(* Logix 5000 project; controller VET 1756-L62 rev 19.52; software revision 19.01 *)

TASK DB (periodic, rate 500 ms, priority 10, watchdog 500 ms) : Main
TASK Dosificador (periodic, rate 40 ms, priority 10, watchdog 250 ms) : Dosificar_MAC_01, Dosificar_MID_01, Dosificar_MIC_01
TASK DRT (periodic, rate 50 ms, priority 1, watchdog 500 ms) : _Ctrl_drt
TASK MainTask (periodic, rate 50 ms, priority 5, watchdog 500 ms) : Main1, Gestion_Dosificacion
TASK Typlgie (periodic, rate 400 ms, priority 10, watchdog 900 ms) : Typlgie

MODULES
   Local : 1756-L62 (ICP 12, rev 19.52)
END_MODULES

TYPE batch :
STRUCT
   Head : batch_cabecera;
   Data : batch_detalle;
END_STRUCT
END_TYPE

TYPE batch_cabecera :
STRUCT
   folio : DINT;
   orden : DINT;
   formula : SHORTSTRING;
   estado : SINT;
   correlativo : SINT;
   total_batch : SINT;
   peso_teorico : REAL;
   flags : SINT;
END_STRUCT
END_TYPE

TYPE batch_detalle :
STRUCT
   codigo : INT[40];   // Código Ingrediente
   peso_f : REAL[40];   // Peso Formula
   peso_r : REAL[40];   // Peso Real
   tolva : SINT[40];   // Tolva Utilizada
   lugar : SINT[40];   // Lugar donde Dosificar
   flags : SINT[40];   // Flags
   fecha_i : DINT[40];
   fecha_f : DINT[40];
   hora_i : DINT[40];
   hora_f : DINT[40];
END_STRUCT
END_TYPE

TYPE Bins_Setup :
STRUCT
   c : tabbin_head;
   d : tabbin_data[2];
END_STRUCT
END_TYPE

TYPE cola_almacenes :
STRUCT
   origen : DINT;
   destino : DINT;
   cantidad : REAL;
   folio_op : DINT;
   fecha : DINT;
   hora : DINT;
END_STRUCT
END_TYPE

TYPE comandos_eph :
STRUCT
   start : BOOL;
   hold : BOOL;
   restart : BOOL;
   stop : BOOL;
   abort : BOOL;
   reset : BOOL;
   reset_especial : BOOL;
END_STRUCT
END_TYPE

TYPE dosif_struct :
STRUCT
   peso_terreno : REAL;
   frq_terreno : REAL;
   idx_ing : INT;
   idx_batch : INT;
   msg : DINT;
   ans : DINT;
   resultado : INT;
   estado_phases : estado_eph;
   comandos_phases : comandos_eph;
END_STRUCT
END_TYPE

TYPE DRTs :   // Estructura para DRT
STRUCT
   InputPos : DINT;   // Posicion Leida (Bits)
   CmdPos : DINT;   // Posicion Comanda
   ConfPos : DINT;   // Posicion Confirmada
   RealPos : DINT;   // Posicion Leida (Num)
   TotalPos : DINT;   // Total Posiciones
END_STRUCT
END_TYPE

TYPE Eqp_Bits :
STRUCT
   Bits1 : DINT;
   Bits2 : DINT;
   Bits3 : DINT;
   Bits4 : DINT;
END_STRUCT
END_TYPE

TYPE Eqp_Cfg :
STRUCT
   Type : DINT;   // Eqp Type
   Setup : DINT;   // Config
   Syst : DINT;   // System Group
   Plant : DINT;   // Plant
   Prst1 : DINT;   // Preset Timer1
   Prst2 : DINT;   // Preset Timer2
   Prst3 : DINT;   // Preset Timer3
   Prst4 : DINT;   // Preset Timer4
   Prst5 : DINT;   // Preset Timer5
   Prst6 : DINT;   // Preset Timer6
END_STRUCT
END_TYPE

TYPE Eqp_Timers :
STRUCT
   Tpo1 : TIMER;
   Tpo2 : TIMER;
   Tpo3 : TIMER;
   Tpo4 : TIMER;
   Tpo5 : TIMER;
   Tpo6 : TIMER;
END_STRUCT
END_TYPE

TYPE Eqp_Typologie :
STRUCT
   Next : DINT;
   Type : DINT;
   Setup : DINT;
   Syst : DINT;
   Area : DINT;
   Indx : DINT[16];
END_STRUCT
END_TYPE

TYPE Equipo :
STRUCT
   Timer : Eqp_Timers;   // Equipment Timers
   S : Eqp_Bits;
   Next : DINT;
   Color : DINT;
END_STRUCT
END_TYPE

TYPE estado_eph :
STRUCT
   _aborted : BOOL;   // Estado Aborted
   _held : BOOL;   // Estado Held
   _idle : BOOL;   // Estado Idle
   _running : BOOL;   // Estado Running
   _complete : BOOL;   // Estado Complete
   _stopped : BOOL;   // Estado Stopped
END_STRUCT
END_TYPE

TYPE falla_aux :
STRUCT
   Time_Low : DINT;
   Time_High : DINT;
   Type : INT;
   Code : INT;
   Info : DINT[8];
   Falla : BOOL;
END_STRUCT
END_TYPE

TYPE Fault_Register :   // Almacena el valor de MAJORFAULTRECORD
STRUCT
   Time_Low : DINT;
   Time_High : DINT;
   Type : INT;
   Code : INT;
   Info : DINT[8];
END_STRUCT
END_TYPE

TYPE flujometro :   // Manejo de Flujometros
STRUCT
   scale_flujo : ScaleAIO;
   scale_total : ScaleAIO;
   flujo : REAL;   // Flujo
   total : REAL;   // Total sin Escalamiento
   total_batch : REAL;   // Peso sin Escalamiento x Batch
   total_scaled : REAL;   // Peso Escalado
   total_scaled_batch : REAL;   // Peso Escalado x Batch
   T : TIMER;
   set_in : REAL;   // Escalamiento Peso Entrada
   set_out : REAL;   // Escalamiento Peso Salida
   aux : DINT;   // Usos Varios
   input : DINT;   // Entrada desde flujómetro
   delta_t : DINT;   // Variación de tiempo en mseg desde la medición anterior
END_STRUCT
END_TYPE

TYPE Index :
STRUCT
   a : DINT;
   b : DINT;
   c : DINT;
   d : DINT;
   e : DINT;
   f : DINT;
   g : DINT;
   h : DINT;
   i : DINT;
   j : DINT;
   k : DINT;
   l : DINT;
   m : DINT;
   n : DINT;
   o : DINT;
   p : DINT;
   q : DINT;
   r : DINT;
   s : DINT;
   t : DINT;
   u : DINT;
   v : DINT;
   w : DINT;
   x : DINT;
   y : DINT;
   z : DINT;
   a1 : DINT;
   b1 : DINT;
   c1 : DINT;
   d1 : DINT;
   e1 : DINT;
   f1 : DINT;
   g1 : DINT;
   h1 : DINT;
   i1 : DINT;
   j1 : DINT;
   k1 : DINT;
   l1 : DINT;
   m1 : DINT;
   n1 : DINT;
   o1 : DINT;
   p1 : DINT;
   q1 : DINT;
   r1 : DINT;
   s1 : DINT;
   t1 : DINT;
   u1 : DINT;
   v1 : DINT;
   w1 : DINT;
   x1 : DINT;
   y1 : DINT;
   z1 : DINT;
   a2 : DINT;
   b2 : DINT;
   c2 : DINT;
   d2 : DINT;
   e2 : DINT;
   f2 : DINT;
   g2 : DINT;
   h2 : DINT;
   i2 : DINT;
   j2 : DINT;
   k2 : DINT;
   l2 : DINT;
   m2 : DINT;
   n2 : DINT;
   o2 : DINT;
   p2 : DINT;
   q2 : DINT;
   r2 : DINT;
   s2 : DINT;
   t2 : DINT;
   u2 : DINT;
   v2 : DINT;
   w2 : DINT;
   x2 : DINT;
   y2 : DINT;
   z2 : DINT;
   a3 : DINT;
   b3 : DINT;
   c3 : DINT;
   d3 : DINT;
   e3 : DINT;
   f3 : DINT;
   g3 : DINT;
   h3 : DINT;
   i3 : DINT;
   j3 : DINT;
   k3 : DINT;
   l3 : DINT;
   m3 : DINT;
   n3 : DINT;
   o3 : DINT;
   p3 : DINT;
   q3 : DINT;
   r3 : DINT;
   s3 : DINT;
   t3 : DINT;
   u3 : DINT;
   v3 : DINT;
   w3 : DINT;
   x3 : DINT;
   y3 : DINT;
   z3 : DINT;
END_STRUCT
END_TYPE

TYPE Origen :
STRUCT
   Index : DINT;   // Index
   _1eqp : DINT;   // Indice Primer Equipo
   Bits : DINT;
   Color : INT;   // Color Linea
   DestReal : DINT;   // Indice Equipo Destino Final Real
   DestOld : DINT;   // Indice Equipo Destino Final Real Old
   DestNew : INT;   // Sub Indice Destino Final
   Prod1eqpInd : DINT;   // Indice Producto Primer Equipo
   ProdFinInd : DINT;   // Indice Producto Bin Final
   Prod1eqp : DINT;   // Codigo Producto Primer Equipo
   ProdFin : DINT;   // Codigo Producto Bin Final
   State : DINT;   // Estado
   Tespera : TIMER;   // Si se cumple este tiempo y no ha partido la ruta se quita la OMR
END_STRUCT
END_TYPE

TYPE PID_Info :
STRUCT
   PV : DINT;   // Process Variable (0-100%)
   SP : DINT;   // Setpoint (0-100%)
   CV : DINT;   // Control Variable (0-100%)
END_STRUCT
END_TYPE

TYPE PID_Struct :
STRUCT
   Core : PID;   // PID Core Instruction
   Status : DINT;   // Status Bits
   Info : PID_Info;   // Extra Information
   PV : REAL;   // Process Variable (ENU)
   SP : REAL;   // Setpoint (ENU)
   CV : REAL;   // Control Variable (0-100%)
   DB : REAL;   // Deadband (ENU)
   Upd : REAL;   // Loop Update Time (sec)
   Kp : REAL;   // Proportional Gain
   Ki : REAL;   // Integral Gain (1/sec)
   Kd : REAL;   // Derivative Time (sec)
   ENU_LL : REAL;   // ENU Low Limit
   ENU_LH : REAL;   // ENU High Limit
   AI : DINT;   // PV - Analog Input (0-4095)
   AO : DINT;   // CV - Analog Output (0-4095)
END_STRUCT
END_TYPE

TYPE Sel_eqp :   // Equipos pertenecientes a selectores
STRUCT
   IDX_SEL : INT;   // Indice Selector al que pertenece
   IDX_EQP : INT;   // Indice Equipo en Tabla Equipos
   POS_CMD : SINT[32];   // Comandos segun posicion
END_STRUCT
END_TYPE

TYPE Selector :
STRUCT
   Idx_eqp : INT;   // Indice en Tabla Equipo
   Next : INT[32];   // Siguiente segun posicion
   Pos_Conf : SINT;   // Posicion Confirmada
   Pos_Cmd : SINT;   // Posicion Comandada
   Pos_Real : SINT;   // Posicion Leida equipos
   Pos_Old : SINT;   // Posicion Anterior RSV
   Pos_New : SINT;   // Posicion Nueva RSV
   Pos_Fut : SINT;   // Posicion Futura RSV
   Pos_Cant : SINT;   // Cantidad de Posiciones
   Pos_CM : SINT;   // Posicion con conf. de marcha
   Idx_1Tabeqp : INT;   // Idx 1er eqp en Tabeqp
   Timer1 : TIMER;
   Timer2 : TIMER;
END_STRUCT
END_TYPE

TYPE set_variables :
STRUCT
   D : DINT[50];
   F : REAL[40];
   T : TIMER[10];
   setD : DINT[10];
   SetF : REAL[10];
   i0 : DINT;
   i1 : DINT;
   i2 : DINT;
   i3 : DINT;
   i4 : DINT;
   i5 : DINT;
   i6 : DINT;
   i7 : DINT;
   i8 : DINT;
   i9 : DINT;
   i10 : DINT;
   i11 : DINT;
   i12 : DINT;
   i13 : DINT;
   i14 : DINT;
   i15 : DINT;
   i16 : DINT;
   i17 : DINT;
   i18 : DINT;
   i19 : DINT;
END_STRUCT
END_TYPE

TYPE SHORTSTRING :
STRUCT
   LEN : DINT;
   DATA : SINT[10];
END_STRUCT
END_TYPE

TYPE Soft_Starter :
STRUCT
   Idx_Equipo : DINT[10];
   Eqp_Actual : DINT;
   Partiendo : BOOL;
   Esperando : BOOL;
   Disponible : BOOL;
   Flags : DINT;
   Procesando : BOOL;
   Tpo_Espera : TIMER;
   Tpos_Grl : TIMER[2];
END_STRUCT
END_TYPE

TYPE STRING12 :
STRUCT
   LEN : DINT;
   DATA : SINT[12];
END_STRUCT
END_TYPE

TYPE STRING14 :
STRUCT
   LEN : DINT;
   DATA : SINT[14];
END_STRUCT
END_TYPE

TYPE Tab_O_D_Dest :
STRUCT
   D : Tab_O_D_Sel[30];   // Destinos Posibles
   Eqp : INT[30];
END_STRUCT
END_TYPE

TYPE Tab_O_D_Orig :
STRUCT
   O : Tab_O_D_Dest[13];   // Numero de Orígnes
END_STRUCT
END_TYPE

TYPE Tab_O_D_Sel :
STRUCT
   S : INT[10];   // NUmero de Selectores
END_STRUCT
END_TYPE

TYPE tabbin_data :
STRUCT
   t_espera : INT[80];   // Tiempo Espera (mSeg)
   t_pulso : INT[80];   // Tiempo Ajuste (mSeg)
   precorte : REAL[80];   // Precorte
   error_per : REAL[80];   // Error Permitido (%)
   error_kg : REAL[80];   // Error Permitido (Kg)
   frec_inicial : REAL[80];   // Frecuencia A (Hz)
   frec_final : REAL[80];   // Frecuencia B (Hz)
   curvatura : REAL[80];   // Curvatura exponencial
   porcentaje_frec_max : REAL[80];   // Porcentaje del peso de detención con dosificación a frecuencia máxima
   low_limit : REAL[80];   // Límite Inferior
   high_limit : REAL[80];   // Límite Superior
   flags : DINT[80];   // Flags Varios
END_STRUCT
END_TYPE

TYPE tabbin_head :
STRUCT
   id : SINT[80];   // Identificador Único de tolva (Correlativo)
   tolva : INT[80];   // Número de Tolva
   n_tolva : DINT[80];   // Número de equipo de la tolva
   equipo1 : INT[80];   // Equipo dosificador
   equipo2 : INT[80];   // Equipo dosificador
   equipo3 : INT[80];   // Equipo dosificador
   equipo4 : INT[80];   // Equipo dosificador
   equipo5 : INT[80];   // Equipo dosificador
   dosificador : INT[80];
   codigo : DINT[80];   // Codigo Ingrediente
   sql_codigo : DINT[80];   // Codigo desde Oracle
   prioridad : INT[80];   // Prioridad
   nivel_bajo : DINT[80];
   nivel_alto : DINT[80];
   tipo : INT[80];
   ind_peso : INT[80];
END_STRUCT
END_TYPE

TYPE tabDosif :   // Tabla de Dosificadores
STRUCT
   idx_tolva : DINT[20];
   idx_vdf : DINT[20];
   idx_flujometro : DINT[20];
   tipo : DINT[20];
END_STRUCT
END_TYPE

TYPE variables_procedimientos :
STRUCT
   step_idx : INT;
   trigger : SINT[5];
   handshake : SINT[5];
   in_tstamp : DINT[5];
   out_tstamp : DINT[5];
   out_res : SINT[5];
   D : DINT[10];
   F : REAL[5];
   i0 : INT;
   i1 : INT;
   i2 : INT;
   i3 : INT;
   i4 : INT;
   SetD : DINT[3];
   SetF : DINT[3];
   T : TIMER[10];
END_STRUCT
END_TYPE

TYPE variables_sproc :
STRUCT
   step_idx : DINT;
   trigger : DINT[3];
   handshake : DINT[3];
   in_tstamp : DINT[3];
   out_tstamp : DINT[3];
   out_res : DINT[3];
   D : DINT[10];
   F : REAL[5];
   i0 : DINT;
   i1 : DINT;
   i2 : DINT;
   i3 : DINT;
   i4 : DINT;
   SetD : DINT[3];
   SetF : DINT[3];
   T : TIMER[5];
END_STRUCT
END_TYPE

TYPE VDFS :
STRUCT
   ST : DINT;
   CMD : DINT;
   FRQ_IN : REAL;
   FRQ_OUT : REAL;
   I : REAL;
   P : REAL;
   V : REAL;
   AUX : DINT[5];
   SCALE : ScaleAIO[2];
   Sincro_MSG : SINT;
END_STRUCT
END_TYPE

ADD_ON_INSTRUCTION ScaleAIO   (* revision 1.0, vendor Ole Bank *)
VAR_INPUT
   Input : REAL; {required}
   InLow : REAL; {required}
   InHigh : REAL; {required}
   OutLow : REAL; {required}
   OutHigh : REAL; {required}
END_VAR
VAR_OUTPUT
   Output : REAL; {access Read Only, required}
END_VAR

ROUTINE Logic   (* ladder *)
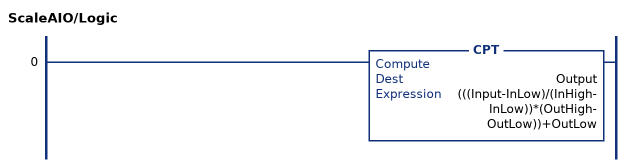
   0: CPT(Output,(((Input-InLow)/(InHigh-InLow))*(OutHigh-OutLow))+OutLow);
END_ROUTINE
END_ADD_ON_INSTRUCTION

ADD_ON_INSTRUCTION velocidad_exp   (* revision 1.0 *)
VAR_INPUT
   x : REAL; {required}
   curvatura : REAL; {required}
   V_inicial : REAL; {required}
   V_final : REAL; {required}
END_VAR
VAR_OUTPUT
   V_salida : REAL; {access Read Only, required}
END_VAR

ROUTINE Logic   (* ladder *)
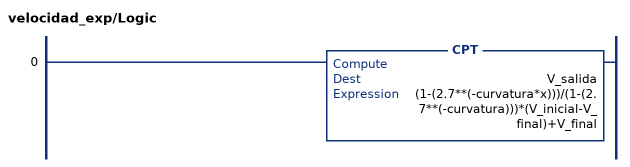
   0: CPT(V_salida,(1-(2.7**(-curvatura*x)))/(1-(2.7**(-curvatura)))*(V_inicial-V_final)+V_final);
END_ROUTINE
END_ADD_ON_INSTRUCTION

VAR_GLOBAL   (* controller tags *)
   _BatCode : DINT[100] := ([0] := 22, [1] := 27, [6] := 17, [28] := 171903600, [29] := 171903600, [30] := 96, [31] := 190628600, [32] := 171680000, [33] := 171903600, [34] := 190628600, [35] := 822086000, [36] := 369524000, [40] := 375774000, [41] := 375774000, [42] := 781952000, [70] := 96);
        [20]   // Codigo DOsificación Macros
        [21]   // Cod. Tolva bajo tolvas pesaje macros
        [31]   // TOL-102-00 Batch
        [32]   // TOL-103-00 Batch
        [33]   // TOL-109-00 Batch
        [34]   // TOL-113-00 Batch
        [36]   // TOL-115-00 Batch
   _Codes : DINT[500] := ([1] := 51, [2] := 51, [3] := 51, [4] := 51, [5] := 51, [6] := 51, [7] := 51, [8] := 51, [9] := 51, [10] := 51, [11] := 51, [12] := 51, [13] := 51, [14] := 51, [15] := 51, [16] := 51, [17] := 51, [18] := 51, [19] := 51, [20] := 51, [21] := 70, [22] := 71, [23] := 72, [24] := 73, [26] := 74, [27] := 75, [28] := 76, [29] := 77, [30] := 78, [31] := 79, [32] := 80, [38] := 81, [101] := 1, [102] := 2, [103] := 3, [104] := 4, [111] := 2, [113] := 2, [200] := 7, [201] := 2238, [202] := 7, [203] := 2081, [204] := 2081, [205] := 2081, [206] := 23, [207] := 23, [209] := 23, [210] := 21, [212] := 23, [214] := 7, [301] := 6706, [302] := 6699, [303] := 6706, [304] := 6707, [305] := 6704, [306] := 6706, [307] := 6703, [309] := 6521, [312] := 6670, [315] := 6675,
        [316] := 6707);
   _Eqp : Equipo[800] := ([1].Timer.Tpo1.PRE := 5000, [1].Timer.Tpo2.PRE := 5000, [1].Timer.Tpo3.PRE := 3000, [1].Timer.Tpo4.PRE := 10000, [1].Timer.Tpo5.PRE := 3000, [1].Timer.Tpo6.PRE := 3000, [1].S.Bits1 := 1, [1].S.Bits2 := 495616, [2].Timer.Tpo1.PRE := 5000, [2].Timer.Tpo2.PRE := 5000, [2].Timer.Tpo3.PRE := 3000, [2].Timer.Tpo4.PRE := 10000, [2].Timer.Tpo5.PRE := 3000, [2].Timer.Tpo6.PRE := 3000, [2].S.Bits1 := 4, [2].S.Bits2 := 1409024, [2].S.Bits3 := 16, [3].Timer.Tpo1.PRE := 5000, [3].Timer.Tpo2.PRE := 5000, [3].Timer.Tpo3.PRE := 3000, [3].Timer.Tpo4.PRE := 10000, [3].Timer.Tpo4.ACC := 10027, [3].Timer.Tpo5.PRE := 3000, [3].Timer.Tpo6.PRE := 3000, [3].S.Bits1 := 65, [3].S.Bits2 := 495616, [3].S.Bits3 := 1073807360, [3].Next := 4, [3].Color := 2, [4].Timer.Tpo1.PRE := 5000, [4].Timer.Tpo2.PRE := 5000, [4].Timer.Tpo3.PRE := 3000, [4].Timer.Tpo4.PRE := 10000, [4].Timer.Tpo4.ACC := 10011, [4].Timer.Tpo5.PRE := 3000, [4].Timer.Tpo6.PRE := 3000, [4].S.Bits1 := 81, [4].S.Bits2 := 2600960, [4].S.Bits3 := 1073807361, [4].Next := 170, [4].Color := 2, [5].Timer.Tpo1.PRE := 5000, [5].Timer.Tpo2.PRE := 5000, [5].Timer.Tpo3.PRE := 3000, [5].Timer.Tpo4.PRE := 10000, [5].Timer.Tpo5.PRE := 3000, [5].Timer.Tpo6.PRE := 3000, [5].S.Bits1 := 1, [5].S.Bits2 := 495616, [6].Timer.Tpo1.PRE := 5000, [6].Timer.Tpo2.PRE := 5000, [6].Timer.Tpo3.PRE := 3000, [6].Timer.Tpo4.PRE := 10000, [6].Timer.Tpo5.PRE := 3000, [6].Timer.Tpo6.PRE := 3000, [6].S.Bits1 := 517, [6].S.Bits2 := 69701635, [7].Timer.Tpo1.PRE := 15000, [7].Timer.Tpo2.PRE := 15000, [7].Timer.Tpo3.PRE := 15000,
        [7].Timer.Tpo4.PRE := 20000, [7].Timer.Tpo5.PRE := 1000, [7].Timer.Tpo6.PRE := 1000, [7].S.Bits1 := 19505, [7].S.Bits2 := 2592768, [8].Timer.Tpo1.PRE := 15000, [8].Timer.Tpo2.PRE := 15000, [8].Timer.Tpo3.PRE := 15000, [8].Timer.Tpo4.PRE := 20000, [8].Timer.Tpo5.PRE := 1000, [8].Timer.Tpo6.PRE := 1000, [8].S.Bits1 := 19505, [8].S.Bits2 := 2592768, [9].Timer.Tpo1.PRE := 5000, [9].Timer.Tpo2.PRE := 5000, [9].Timer.Tpo3.PRE := 3000, [9].Timer.Tpo4.PRE := 10000, [9].Timer.Tpo5.PRE := 3000, [9].Timer.Tpo6.PRE := 3000, [10].Timer.Tpo1.PRE := 10000, [10].Timer.Tpo2.PRE := 10000, [10].Timer.Tpo3.PRE := 10000, [10].Timer.Tpo4.PRE := 10000, [10].Timer.Tpo5.PRE := 3000, [10].Timer.Tpo6.PRE := 3000, [10].S.Bits1 := 593, [10].S.Bits2 := 2600960, [10].S.Bits3 := 1073807361, [10].Next := 110, [10].Color := 2, [11].Timer.Tpo1.PRE := 5000, [11].Timer.Tpo2.PRE := 5000, [11].Timer.Tpo3.PRE := 3000, [11].Timer.Tpo4.PRE := 10000, [11].Timer.Tpo5.PRE := 3000, [11].Timer.Tpo6.PRE := 3000, [11].S.Bits1 := 593, [11].S.Bits2 := 2600960, [11].S.Bits3 := 1073807361, [11].Next := 112, [11].Color := 2, [12].Timer.Tpo1.PRE := 5000, [12].Timer.Tpo2.PRE := 5000, [12].Timer.Tpo3.PRE := 3000, [12].Timer.Tpo4.PRE := 45000, [12].Timer.Tpo5.PRE := 15000, [12].Timer.Tpo6.PRE := 3000, [12].S.Bits1 := 593, [12].S.Bits2 := 2600960, [12].S.Bits3 := 1073807361, [12].Next := 112, [12].Color := 2, [13].Timer.Tpo1.PRE := 5000, [13].Timer.Tpo2.PRE := 5000, [13].Timer.Tpo3.PRE := 3000, [13].Timer.Tpo4.PRE := 10000, [13].Timer.Tpo5.PRE := 3000, [13].Timer.Tpo6.PRE := 3000, [13].S.Bits1 := 593, [13].S.Bits2 := 2600960,
        [13].S.Bits3 := 1073807361, [13].Next := 110, [13].Color := 2, [14].Timer.Tpo1.PRE := 5000, [14].Timer.Tpo2.PRE := 5000, [14].Timer.Tpo3.PRE := 3000, [14].Timer.Tpo4.PRE := 10000, [14].Timer.Tpo5.PRE := 3000, [14].Timer.Tpo6.PRE := 3000, [14].S.Bits1 := 593, [14].S.Bits2 := 2600960, [14].S.Bits3 := 1073807361, [14].Next := 110, [14].Color := 2, [15].Timer.Tpo1.PRE := 5000, [15].Timer.Tpo2.PRE := 5000, [15].Timer.Tpo3.PRE := 3000, [15].Timer.Tpo4.PRE := 10000, [15].Timer.Tpo5.PRE := 3000, [15].Timer.Tpo6.PRE := 3000, [15].S.Bits1 := 593, [15].S.Bits2 := 2600960, [15].S.Bits3 := 1073807361, [15].Next := 112, [15].Color := 2, [16].Timer.Tpo1.PRE := 5000, [16].Timer.Tpo2.PRE := 5000, [16].Timer.Tpo3.PRE := 3000, [16].Timer.Tpo4.PRE := 10000, [16].Timer.Tpo5.PRE := 3000, [16].Timer.Tpo6.PRE := 3000, [17].Timer.Tpo1.PRE := 5000, [17].Timer.Tpo2.PRE := 5000, [17].Timer.Tpo3.PRE := 3000, [17].Timer.Tpo4.PRE := 10000, [17].Timer.Tpo5.PRE := 3000, [17].Timer.Tpo6.PRE := 3000, [18].Timer.Tpo1.PRE := 5000, [18].Timer.Tpo2.PRE := 5000, [18].Timer.Tpo3.PRE := 3000, [18].Timer.Tpo4.PRE := 10000, [18].Timer.Tpo5.PRE := 3000, [18].Timer.Tpo6.PRE := 3000, [19].Timer.Tpo1.PRE := 5000, [19].Timer.Tpo2.PRE := 5000, [19].Timer.Tpo3.PRE := 3000, [19].Timer.Tpo4.PRE := 10000, [19].Timer.Tpo5.PRE := 3000, [19].Timer.Tpo6.PRE := 3000, [20].Timer.Tpo1.PRE := 5000, [20].Timer.Tpo2.PRE := 5000, [20].Timer.Tpo3.PRE := 3000, [20].Timer.Tpo4.PRE := 10000, [20].Timer.Tpo5.PRE := 3000, [20].Timer.Tpo6.PRE := 3000, [20].S.Bits1 := 4, [20].S.Bits2 := 1409024, [20].S.Bits3 := 16, [21].Timer.Tpo1.PRE := 5000, [21].Timer.Tpo2.PRE := 5000,
        [21].Timer.Tpo3.PRE := 3000, [21].Timer.Tpo4.PRE := 10000, [21].Timer.Tpo5.PRE := 3000, [21].Timer.Tpo6.PRE := 3000, [21].S.Bits1 := 4, [21].S.Bits2 := 1409024, [21].S.Bits3 := 16, [22].Timer.Tpo1.PRE := 5000, [22].Timer.Tpo2.PRE := 5000, [22].Timer.Tpo3.PRE := 3000, [22].Timer.Tpo4.PRE := 45000, [22].Timer.Tpo5.PRE := 15000, [22].Timer.Tpo6.PRE := 3000, [22].S.Bits1 := 4, [22].S.Bits2 := 1409024, [22].S.Bits3 := 16, [23].Timer.Tpo1.PRE := 5000, [23].Timer.Tpo2.PRE := 5000, [23].Timer.Tpo3.PRE := 3000, [23].Timer.Tpo4.PRE := 10000, [23].Timer.Tpo5.PRE := 3000, [23].Timer.Tpo6.PRE := 3000, [23].S.Bits1 := 4, [23].S.Bits2 := 1409024, [23].S.Bits3 := 16, [24].Timer.Tpo1.PRE := 5000, [24].Timer.Tpo2.PRE := 5000, [24].Timer.Tpo3.PRE := 3000, [24].Timer.Tpo4.PRE := 10000, [24].Timer.Tpo5.PRE := 3000, [24].Timer.Tpo6.PRE := 3000, [24].S.Bits1 := 4, [24].S.Bits2 := 1409024, [24].S.Bits3 := 16, [25].Timer.Tpo1.PRE := 5000, [25].Timer.Tpo2.PRE := 5000, [25].Timer.Tpo3.PRE := 3000, [25].Timer.Tpo4.PRE := 10000, [25].Timer.Tpo5.PRE := 3000, [25].Timer.Tpo6.PRE := 3000, [25].S.Bits1 := 4, [25].S.Bits2 := 1409024, [25].S.Bits3 := 16, [26].Timer.Tpo1.PRE := 5000, [26].Timer.Tpo2.PRE := 5000, [26].Timer.Tpo3.PRE := 3000, [26].Timer.Tpo4.PRE := 10000, [26].Timer.Tpo5.PRE := 3000, [26].Timer.Tpo6.PRE := 3000, [26].S.Bits1 := 4, [26].S.Bits2 := 1409024, [26].S.Bits3 := 16, [27].Timer.Tpo1.PRE := 5000, [27].Timer.Tpo2.PRE := 5000, [27].Timer.Tpo3.PRE := 3000, [27].Timer.Tpo4.PRE := 10000, [27].Timer.Tpo5.PRE := 3000, [27].Timer.Tpo6.PRE := 3000, [27].S.Bits1 := 4, [27].S.Bits2 := 1409024,
        [27].S.Bits3 := 16, [28].Timer.Tpo1.PRE := 5000, [28].Timer.Tpo2.PRE := 5000, [28].Timer.Tpo3.PRE := 3000, [28].Timer.Tpo4.PRE := 10000, [28].Timer.Tpo5.PRE := 3000, [28].Timer.Tpo6.PRE := 3000, [28].S.Bits1 := 4, [28].S.Bits2 := 1409024, [28].S.Bits3 := 16, [29].Timer.Tpo1.PRE := 5000, [29].Timer.Tpo2.PRE := 5000, [29].Timer.Tpo3.PRE := 3000, [29].Timer.Tpo4.PRE := 10000, [29].Timer.Tpo5.PRE := 3000, [29].Timer.Tpo6.PRE := 3000, [29].S.Bits1 := 4, [29].S.Bits2 := 1409024, [29].S.Bits3 := 16, [30].Timer.Tpo1.PRE := 5000, [30].Timer.Tpo2.PRE := 5000, [30].Timer.Tpo3.PRE := 3000, [30].Timer.Tpo4.PRE := 10000, [30].Timer.Tpo5.PRE := 3000, [30].Timer.Tpo6.PRE := 3000, [30].S.Bits1 := 4, [30].S.Bits2 := 1409024, [30].S.Bits3 := 16, [31].Timer.Tpo1.PRE := 5000, [31].Timer.Tpo2.PRE := 5000, [31].Timer.Tpo3.PRE := 3000, [31].Timer.Tpo4.PRE := 10000, [31].Timer.Tpo5.PRE := 3000, [31].Timer.Tpo6.PRE := 3000, [31].S.Bits1 := 4, [31].S.Bits2 := 1409024, [31].S.Bits3 := 16, [32].Timer.Tpo1.PRE := 5000, [32].Timer.Tpo2.PRE := 5000, [32].Timer.Tpo3.PRE := 3000, [32].Timer.Tpo4.PRE := 10000, [32].Timer.Tpo5.PRE := 3000, [32].Timer.Tpo6.PRE := 3000, [32].S.Bits1 := 4, [32].S.Bits2 := 1409024, [32].S.Bits3 := 16, [33].Timer.Tpo1.PRE := 5000, [33].Timer.Tpo2.PRE := 5000, [33].Timer.Tpo3.PRE := 3000, [33].Timer.Tpo4.PRE := 10000, [33].Timer.Tpo5.PRE := 3000, [33].Timer.Tpo6.PRE := 3000, [33].S.Bits1 := 4, [33].S.Bits2 := 1409024, [33].S.Bits3 := 16, [34].Timer.Tpo1.PRE := 5000, [34].Timer.Tpo2.PRE := 5000, [34].Timer.Tpo3.PRE := 3000, [34].Timer.Tpo4.PRE := 10000, [34].Timer.Tpo5.PRE := 3000,
        [34].Timer.Tpo6.PRE := 3000, [34].S.Bits1 := 4, [34].S.Bits2 := 1409024, [34].S.Bits3 := 16, [35].Timer.Tpo1.PRE := 5000, [35].Timer.Tpo2.PRE := 5000, [35].Timer.Tpo3.PRE := 3000, [35].Timer.Tpo4.PRE := 10000, [35].Timer.Tpo5.PRE := 3000, [35].Timer.Tpo6.PRE := 3000, [35].S.Bits1 := 4, [35].S.Bits2 := 1409024, [35].S.Bits3 := 16, [36].Timer.Tpo1.PRE := 5000, [36].Timer.Tpo2.PRE := 5000, [36].Timer.Tpo3.PRE := 3000, [36].Timer.Tpo4.PRE := 10000, [36].Timer.Tpo5.PRE := 3000, [36].Timer.Tpo6.PRE := 3000, [37].Timer.Tpo1.PRE := 5000, [37].Timer.Tpo2.PRE := 5000, [37].Timer.Tpo3.PRE := 3000, [37].Timer.Tpo4.PRE := 10000, [37].Timer.Tpo5.PRE := 3000, [37].Timer.Tpo6.PRE := 3000, [38].Timer.Tpo1.PRE := 5000, [38].Timer.Tpo2.PRE := 5000, [38].Timer.Tpo3.PRE := 3000, [38].Timer.Tpo4.PRE := 10000, [38].Timer.Tpo5.PRE := 3000, [38].Timer.Tpo6.PRE := 3000, [39].Timer.Tpo1.PRE := 5000, [39].Timer.Tpo2.PRE := 5000, [39].Timer.Tpo3.PRE := 3000, [39].Timer.Tpo4.PRE := 10000, [39].Timer.Tpo5.PRE := 3000, [39].Timer.Tpo6.PRE := 3000, [40].Timer.Tpo1.PRE := 5000, [40].Timer.Tpo2.PRE := 5000, [40].Timer.Tpo3.PRE := 3000, [40].Timer.Tpo4.PRE := 10000, [40].Timer.Tpo5.PRE := 3000, [40].Timer.Tpo6.PRE := 3000, [40].S.Bits1 := 81, [40].S.Bits2 := 2600960, [40].S.Bits3 := 1073807361, [40].Next := 110, [40].Color := 2, [41].Timer.Tpo1.PRE := 5000, [41].Timer.Tpo2.PRE := 5000, [41].Timer.Tpo3.PRE := 3000, [41].Timer.Tpo4.PRE := 10000, [41].Timer.Tpo5.PRE := 3000, [41].Timer.Tpo6.PRE := 3000, [41].S.Bits1 := 81, [41].S.Bits2 := 2600960, [41].S.Bits3 := 1073807361, [41].Next := 110, [41].Color := 2, [42].Timer.Tpo1.PRE := 5000,
        [42].Timer.Tpo2.PRE := 5000, [42].Timer.Tpo3.PRE := 3000, [42].Timer.Tpo4.PRE := 10000, [42].Timer.Tpo5.PRE := 3000, [42].Timer.Tpo6.PRE := 3000, [42].S.Bits1 := 81, [42].S.Bits2 := 2600960, [42].S.Bits3 := 1073807361, [42].Next := 110, [42].Color := 2, [43].Timer.Tpo1.PRE := 5000, [43].Timer.Tpo2.PRE := 5000, [43].Timer.Tpo3.PRE := 3000, [43].Timer.Tpo4.PRE := 10000, [43].Timer.Tpo5.PRE := 3000, [43].Timer.Tpo6.PRE := 3000, [43].S.Bits1 := 65, [43].S.Bits2 := 495616, [43].S.Bits3 := 1073807360, [43].Next := 10, [43].Color := 2, [44].Timer.Tpo1.PRE := 5000, [44].Timer.Tpo2.PRE := 5000, [44].Timer.Tpo3.PRE := 3000, [44].Timer.Tpo4.PRE := 10000, [44].Timer.Tpo5.PRE := 3000, [44].Timer.Tpo6.PRE := 3000, [44].S.Bits1 := 65, [44].S.Bits2 := 495616, [44].S.Bits3 := 1073807360, [44].Next := 11, [44].Color := 2, [45].Timer.Tpo1.PRE := 5000, [45].Timer.Tpo2.PRE := 5000, [45].Timer.Tpo3.PRE := 3000, [45].Timer.Tpo5.PRE := 3000, [45].Timer.Tpo6.PRE := 3000, [45].S.Bits1 := 81, [45].S.Bits2 := 2600960, [45].S.Bits3 := 1073807361, [45].Next := 112, [45].Color := 2, [46].Timer.Tpo1.PRE := 5000, [46].Timer.Tpo2.PRE := 5000, [46].Timer.Tpo3.PRE := 3000, [46].Timer.Tpo5.PRE := 3000, [46].Timer.Tpo6.PRE := 3000, [46].S.Bits1 := 65, [46].S.Bits2 := 495616, [46].S.Bits3 := 1073807360, [46].Next := 12, [46].Color := 2, [47].Timer.Tpo1.PRE := 5000, [47].Timer.Tpo2.PRE := 5000, [47].Timer.Tpo3.PRE := 3000, [47].Timer.Tpo4.PRE := 10000, [47].Timer.Tpo5.PRE := 5000, [47].Timer.Tpo6.PRE := 3000, [47].S.Bits1 := 81, [47].S.Bits2 := 2600960,
        [47].S.Bits3 := 1073807361, [47].Next := 112, [47].Color := 2, [48].Timer.Tpo1.PRE := 5000, [48].Timer.Tpo2.PRE := 5000, [48].Timer.Tpo3.PRE := 3000, [48].Timer.Tpo4.PRE := 10000, [48].Timer.Tpo5.PRE := 5000, [48].Timer.Tpo6.PRE := 3000, [48].S.Bits1 := 81, [48].S.Bits2 := 2600960, [48].S.Bits3 := 1073807361, [48].Next := 110, [48].Color := 2, [49].Timer.Tpo1.PRE := 5000, [49].Timer.Tpo2.PRE := 5000, [49].Timer.Tpo3.PRE := 3000, [49].Timer.Tpo4.PRE := 10000, [49].Timer.Tpo5.PRE := 3000, [49].Timer.Tpo6.PRE := 3000, [49].S.Bits1 := 65, [49].S.Bits2 := 495616, [49].S.Bits3 := 1073807360, [49].Next := 13, [49].Color := 2, [50].Timer.Tpo1.PRE := 5000, [50].Timer.Tpo2.PRE := 5000, [50].Timer.Tpo3.PRE := 3000, [50].Timer.Tpo4.PRE := 10000, [50].Timer.Tpo5.PRE := 3000, [50].Timer.Tpo6.PRE := 15000, [50].S.Bits1 := 81, [50].S.Bits2 := 2600960, [50].S.Bits3 := 1073807361, [50].Next := 110, [50].Color := 2, [51].Timer.Tpo1.PRE := 5000, [51].Timer.Tpo2.PRE := 5000, [51].Timer.Tpo3.PRE := 3000, [51].Timer.Tpo4.PRE := 10000, [51].Timer.Tpo5.PRE := 3000, [51].Timer.Tpo6.PRE := 3000, [51].S.Bits1 := 65, [51].S.Bits2 := 495616, [51].S.Bits3 := 1073807360, [51].Next := 14, [51].Color := 2, [52].Timer.Tpo1.PRE := 5000, [52].Timer.Tpo2.PRE := 5000, [52].Timer.Tpo3.PRE := 3000, [52].Timer.Tpo4.PRE := 10000, [52].Timer.Tpo5.PRE := 3000, [52].Timer.Tpo6.PRE := 3000, [52].S.Bits1 := 81, [52].S.Bits2 := 2600960, [52].S.Bits3 := 1073807361, [52].Next := 112, [52].Color := 2, [53].Timer.Tpo1.PRE := 5000, [53].Timer.Tpo2.PRE := 5000,
        [53].Timer.Tpo3.PRE := 3000, [53].Timer.Tpo4.PRE := 10000, [53].Timer.Tpo5.PRE := 3000, [53].Timer.Tpo6.PRE := 3000, [53].S.Bits1 := 81, [53].S.Bits2 := 2600960, [53].S.Bits3 := 1073807361, [53].Next := 112, [53].Color := 2, [54].Timer.Tpo1.PRE := 5000, [54].Timer.Tpo2.PRE := 5000, [54].Timer.Tpo3.PRE := 3000, [54].Timer.Tpo4.PRE := 10000, [54].Timer.Tpo5.PRE := 3000, [54].Timer.Tpo6.PRE := 3000, [54].S.Bits1 := 81, [54].S.Bits2 := 2600960, [54].S.Bits3 := 1073807361, [54].Next := 112, [54].Color := 2, [55].Timer.Tpo1.PRE := 5000, [55].Timer.Tpo2.PRE := 5000, [55].Timer.Tpo3.PRE := 3000, [55].Timer.Tpo4.PRE := 10000, [55].Timer.Tpo5.PRE := 3000, [55].Timer.Tpo6.PRE := 3000, [55].S.Bits1 := 65, [55].S.Bits2 := 495616, [55].S.Bits3 := 1073807360, [55].Next := 15, [55].Color := 2, [56].Timer.Tpo1.PRE := 5000, [56].Timer.Tpo2.PRE := 5000, [56].Timer.Tpo3.PRE := 3000, [56].Timer.Tpo4.PRE := 10000, [56].Timer.Tpo5.PRE := 3000, [56].Timer.Tpo6.PRE := 3000, [57].Timer.Tpo1.PRE := 5000, [57].Timer.Tpo2.PRE := 5000, [57].Timer.Tpo3.PRE := 3000, [57].Timer.Tpo5.PRE := 3000, [57].Timer.Tpo6.PRE := 3000, [58].Timer.Tpo1.PRE := 5000, [58].Timer.Tpo2.PRE := 5000, [58].Timer.Tpo3.PRE := 3000, [58].Timer.Tpo5.PRE := 3000, [58].Timer.Tpo6.PRE := 3000, [59].Timer.Tpo1.PRE := 5000, [59].Timer.Tpo2.PRE := 5000, [59].Timer.Tpo3.PRE := 3000, [59].Timer.Tpo4.PRE := 10000, [59].Timer.Tpo5.PRE := 5000, [59].Timer.Tpo6.PRE := 3000, [60].Timer.Tpo1.PRE := 5000, [60].Timer.Tpo2.PRE := 5000, [60].Timer.Tpo3.PRE := 3000, [60].Timer.Tpo4.PRE := 10000, [60].Timer.Tpo5.PRE := 5000, [60].Timer.Tpo6.PRE := 3000, [60].S.Bits1 := 4,
        [60].S.Bits2 := 1409024, [60].S.Bits3 := 16, [61].Timer.Tpo1.PRE := 5000, [61].Timer.Tpo2.PRE := 5000, [61].Timer.Tpo3.PRE := 3000, [61].Timer.Tpo4.PRE := 10000, [61].Timer.Tpo5.PRE := 3000, [61].Timer.Tpo6.PRE := 3000, [61].S.Bits1 := 4, [61].S.Bits2 := 1409024, [61].S.Bits3 := 16, [62].Timer.Tpo1.PRE := 5000, [62].Timer.Tpo2.PRE := 5000, [62].Timer.Tpo3.PRE := 3000, [62].Timer.Tpo4.PRE := 10000, [62].Timer.Tpo5.PRE := 3000, [62].Timer.Tpo6.PRE := 15000, [62].S.Bits1 := 4, [62].S.Bits2 := 1409024, [62].S.Bits3 := 16, [63].Timer.Tpo1.PRE := 5000, [63].Timer.Tpo2.PRE := 5000, [63].Timer.Tpo3.PRE := 3000, [63].Timer.Tpo4.PRE := 10000, [63].Timer.Tpo5.PRE := 3000, [63].Timer.Tpo6.PRE := 3000, [63].S.Bits1 := 4, [63].S.Bits2 := 1409024, [63].S.Bits3 := 16, [64].Timer.Tpo1.PRE := 5000, [64].Timer.Tpo2.PRE := 5000, [64].Timer.Tpo3.PRE := 3000, [64].Timer.Tpo4.PRE := 10000, [64].Timer.Tpo5.PRE := 3000, [64].Timer.Tpo6.PRE := 3000, [64].S.Bits1 := 4, [64].S.Bits2 := 1409024, [64].S.Bits3 := 16, [65].Timer.Tpo1.PRE := 5000, [65].Timer.Tpo2.PRE := 5000, [65].Timer.Tpo3.PRE := 3000, [65].Timer.Tpo4.PRE := 10000, [65].Timer.Tpo5.PRE := 3000, [65].Timer.Tpo6.PRE := 3000, [65].S.Bits1 := 4, [65].S.Bits2 := 1409024, [65].S.Bits3 := 16, [66].Timer.Tpo1.PRE := 5000, [66].Timer.Tpo2.PRE := 5000, [66].Timer.Tpo3.PRE := 3000, [66].Timer.Tpo4.PRE := 10000, [66].Timer.Tpo5.PRE := 3000, [66].Timer.Tpo6.PRE := 3000, [66].S.Bits1 := 4, [66].S.Bits2 := 1409024, [66].S.Bits3 := 16, [67].Timer.Tpo1.PRE := 5000, [67].Timer.Tpo2.PRE := 5000, [67].Timer.Tpo3.PRE := 3000, [67].Timer.Tpo4.PRE := 10000,
        [67].Timer.Tpo5.PRE := 3000, [67].Timer.Tpo6.PRE := 3000, [67].S.Bits1 := 4, [67].S.Bits2 := 1409024, [67].S.Bits3 := 16, [68].Timer.Tpo1.PRE := 5000, [68].Timer.Tpo2.PRE := 5000, [68].Timer.Tpo3.PRE := 3000, [68].Timer.Tpo4.PRE := 10000, [68].Timer.Tpo5.PRE := 3000, [68].Timer.Tpo6.PRE := 3000, [68].S.Bits1 := 4, [68].S.Bits2 := 1409024, [68].S.Bits3 := 16, [69].Timer.Tpo1.PRE := 5000, [69].Timer.Tpo2.PRE := 5000, [69].Timer.Tpo3.PRE := 3000, [69].Timer.Tpo5.PRE := 3000, [69].Timer.Tpo6.PRE := 3000, [69].S.Bits1 := 4, [69].S.Bits2 := 1409024, [69].S.Bits3 := 16, [70].Timer.Tpo1.PRE := 5000, [70].Timer.Tpo2.PRE := 5000, [70].Timer.Tpo3.PRE := 3000, [70].Timer.Tpo5.PRE := 3000, [70].Timer.Tpo6.PRE := 3000, [70].S.Bits1 := 4, [70].S.Bits2 := 1409024, [70].S.Bits3 := 16, [71].Timer.Tpo1.PRE := 5000, [71].Timer.Tpo2.PRE := 5000, [71].Timer.Tpo3.PRE := 3000, [71].Timer.Tpo4.PRE := 10000, [71].Timer.Tpo5.PRE := 5000, [71].Timer.Tpo6.PRE := 3000, [71].S.Bits1 := 4, [71].S.Bits2 := 1409024, [71].S.Bits3 := 16, [72].Timer.Tpo1.PRE := 5000, [72].Timer.Tpo2.PRE := 5000, [72].Timer.Tpo3.PRE := 3000, [72].Timer.Tpo4.PRE := 10000, [72].Timer.Tpo5.PRE := 5000, [72].Timer.Tpo6.PRE := 3000, [72].S.Bits1 := 4, [72].S.Bits2 := 1409024, [72].S.Bits3 := 16, [73].Timer.Tpo1.PRE := 5000, [73].Timer.Tpo2.PRE := 5000, [73].Timer.Tpo3.PRE := 3000, [73].Timer.Tpo4.PRE := 10000, [73].Timer.Tpo5.PRE := 3000, [73].Timer.Tpo6.PRE := 3000, [73].S.Bits1 := 4, [73].S.Bits2 := 1409024, [73].S.Bits3 := 16, [74].Timer.Tpo1.PRE := 5000, [74].Timer.Tpo2.PRE := 5000, [74].Timer.Tpo3.PRE := 3000,
        [74].Timer.Tpo4.PRE := 10000, [74].Timer.Tpo5.PRE := 3000, [74].Timer.Tpo6.PRE := 15000, [74].S.Bits1 := 4, [74].S.Bits2 := 1409024, [74].Next := 94, [75].Timer.Tpo1.PRE := 5000, [75].Timer.Tpo2.PRE := 5000, [75].Timer.Tpo3.PRE := 3000, [75].Timer.Tpo4.PRE := 10000, [75].Timer.Tpo5.PRE := 3000, [75].Timer.Tpo6.PRE := 3000, [76].Timer.Tpo1.PRE := 5000, [76].Timer.Tpo2.PRE := 5000, [76].Timer.Tpo3.PRE := 3000, [76].Timer.Tpo4.PRE := 10000, [76].Timer.Tpo5.PRE := 3000, [76].Timer.Tpo6.PRE := 3000, [77].Timer.Tpo1.PRE := 5000, [77].Timer.Tpo2.PRE := 5000, [77].Timer.Tpo3.PRE := 3000, [77].Timer.Tpo4.PRE := 10000, [77].Timer.Tpo5.PRE := 3000, [77].Timer.Tpo6.PRE := 3000, [78].Timer.Tpo1.PRE := 5000, [78].Timer.Tpo2.PRE := 5000, [78].Timer.Tpo3.PRE := 3000, [78].Timer.Tpo4.PRE := 10000, [78].Timer.Tpo5.PRE := 3000, [78].Timer.Tpo6.PRE := 3000, [79].Timer.Tpo1.PRE := 5000, [79].Timer.Tpo2.PRE := 5000, [79].Timer.Tpo3.PRE := 3000, [79].Timer.Tpo4.PRE := 10000, [79].Timer.Tpo5.PRE := 3000, [79].Timer.Tpo6.PRE := 3000, [80].Timer.Tpo1.PRE := 5000, [80].Timer.Tpo2.PRE := 5000, [80].Timer.Tpo3.PRE := 3000, [80].Timer.Tpo4.PRE := 10000, [80].Timer.Tpo5.PRE := 3000, [80].Timer.Tpo6.PRE := 3000, [80].S.Bits1 := 81, [80].S.Bits2 := 2600960, [80].S.Bits3 := 1073807361, [80].Next := 114, [80].Color := 2, [81].Timer.Tpo1.PRE := 5000, [81].Timer.Tpo2.PRE := 5000, [81].Timer.Tpo3.PRE := 3000, [81].Timer.Tpo5.PRE := 3000, [81].Timer.Tpo6.PRE := 3000, [81].S.Bits1 := 65, [81].S.Bits2 := 495616, [81].S.Bits3 := 1073807360, [81].Next := 100, [81].Color := 2, [82].Timer.Tpo1.PRE := 5000, [82].Timer.Tpo2.PRE := 5000, [82].Timer.Tpo3.PRE := 3000,
        [82].Timer.Tpo5.PRE := 3000, [82].Timer.Tpo6.PRE := 3000, [82].S.Bits1 := 81, [82].S.Bits2 := 2600960, [82].S.Bits3 := 1073807361, [82].Next := 114, [82].Color := 2, [83].Timer.Tpo1.PRE := 5000, [83].Timer.Tpo2.PRE := 5000, [83].Timer.Tpo3.PRE := 3000, [83].Timer.Tpo4.PRE := 10000, [83].Timer.Tpo5.PRE := 5000, [83].Timer.Tpo6.PRE := 3000, [83].S.Bits1 := 65, [83].S.Bits2 := 495616, [83].S.Bits3 := 1073807360, [83].Next := 101, [83].Color := 2, [84].Timer.Tpo1.PRE := 5000, [84].Timer.Tpo2.PRE := 5000, [84].Timer.Tpo3.PRE := 3000, [84].Timer.Tpo4.PRE := 10000, [84].Timer.Tpo5.PRE := 5000, [84].Timer.Tpo6.PRE := 3000, [84].S.Bits1 := 81, [84].S.Bits2 := 2600960, [84].S.Bits3 := 1073807361, [84].Next := 114, [84].Color := 2, [85].Timer.Tpo1.PRE := 5000, [85].Timer.Tpo2.PRE := 5000, [85].Timer.Tpo3.PRE := 3000, [85].Timer.Tpo4.PRE := 10000, [85].Timer.Tpo5.PRE := 3000, [85].Timer.Tpo6.PRE := 3000, [85].S.Bits1 := 65, [85].S.Bits2 := 495616, [85].S.Bits3 := 1073807360, [85].Next := 102, [85].Color := 2, [86].Timer.Tpo1.PRE := 5000, [86].Timer.Tpo2.PRE := 5000, [86].Timer.Tpo3.PRE := 3000, [86].Timer.Tpo4.PRE := 10000, [86].Timer.Tpo5.PRE := 3000, [86].Timer.Tpo6.PRE := 15000, [86].S.Bits1 := 81, [86].S.Bits2 := 2600960, [86].S.Bits3 := 1073807361, [86].Next := 114, [86].Color := 2, [87].Timer.Tpo1.PRE := 5000, [87].Timer.Tpo2.PRE := 5000, [87].Timer.Tpo3.PRE := 3000, [87].Timer.Tpo4.PRE := 10000, [87].Timer.Tpo5.PRE := 3000, [87].Timer.Tpo6.PRE := 3000, [87].S.Bits1 := 81, [87].S.Bits2 := 2600960, [87].S.Bits3 := 1073807361,
        [87].Next := 116, [87].Color := 2, [88].Timer.Tpo1.PRE := 5000, [88].Timer.Tpo2.PRE := 5000, [88].Timer.Tpo3.PRE := 3000, [88].Timer.Tpo4.PRE := 10000, [88].Timer.Tpo5.PRE := 3000, [88].Timer.Tpo6.PRE := 3000, [88].S.Bits1 := 65, [88].S.Bits2 := 495616, [88].S.Bits3 := 1073807360, [88].Next := 103, [88].Color := 2, [89].Timer.Tpo1.PRE := 5000, [89].Timer.Tpo2.PRE := 5000, [89].Timer.Tpo3.PRE := 3000, [89].Timer.Tpo4.PRE := 10000, [89].Timer.Tpo5.PRE := 3000, [89].Timer.Tpo6.PRE := 3000, [89].S.Bits1 := 81, [89].S.Bits2 := 2600960, [89].S.Bits3 := 1073807361, [89].Next := 116, [89].Color := 2, [90].Timer.Tpo1.PRE := 5000, [90].Timer.Tpo2.PRE := 5000, [90].Timer.Tpo3.PRE := 3000, [90].Timer.Tpo4.PRE := 10000, [90].Timer.Tpo5.PRE := 3000, [90].Timer.Tpo6.PRE := 3000, [90].S.Bits1 := 65, [90].S.Bits2 := 495616, [90].S.Bits3 := 1073807360, [90].Next := 104, [90].Color := 2, [91].Timer.Tpo1.PRE := 5000, [91].Timer.Tpo2.PRE := 5000, [91].Timer.Tpo3.PRE := 3000, [91].Timer.Tpo4.PRE := 10000, [91].Timer.Tpo5.PRE := 3000, [91].Timer.Tpo6.PRE := 3000, [91].S.Bits1 := 81, [91].S.Bits2 := 2600960, [91].S.Bits3 := 1073807361, [91].Next := 116, [91].Color := 2, [92].Timer.Tpo1.PRE := 5000, [92].Timer.Tpo2.PRE := 5000, [92].Timer.Tpo3.PRE := 3000, [92].Timer.Tpo4.PRE := 10000, [92].Timer.Tpo5.PRE := 3000, [92].Timer.Tpo6.PRE := 3000, [92].S.Bits1 := 65, [92].S.Bits2 := 495616, [92].S.Bits3 := 1073807360, [92].Next := 105, [92].Color := 2, [93].Timer.Tpo1.PRE := 5000, [93].Timer.Tpo2.PRE := 5000, [93].Timer.Tpo3.PRE := 3000,
        [93].Timer.Tpo5.PRE := 3000, [93].Timer.Tpo6.PRE := 3000, [93].S.Bits1 := 81, [93].S.Bits2 := 2600960, [93].S.Bits3 := 1073807361, [93].Next := 116, [93].Color := 2, [94].Timer.Tpo1.PRE := 5000, [94].Timer.Tpo2.PRE := 5000, [94].Timer.Tpo3.PRE := 3000, [94].Timer.Tpo5.PRE := 3000, [94].Timer.Tpo6.PRE := 3000, [94].S.Bits1 := 593, [94].S.Bits2 := 495616, [94].S.Bits3 := 1073807360, [94].Next := 119, [94].Color := 2, [95].Timer.Tpo1.PRE := 5000, [95].Timer.Tpo2.PRE := 5000, [95].Timer.Tpo3.PRE := 3000, [95].Timer.Tpo4.PRE := 10000, [95].Timer.Tpo5.PRE := 5000, [95].Timer.Tpo6.PRE := 3000, [96].Timer.Tpo1.PRE := 5000, [96].Timer.Tpo2.PRE := 5000, [96].Timer.Tpo3.PRE := 3000, [96].Timer.Tpo4.PRE := 10000, [96].Timer.Tpo5.PRE := 5000, [96].Timer.Tpo6.PRE := 3000, [97].Timer.Tpo1.PRE := 5000, [97].Timer.Tpo2.PRE := 5000, [97].Timer.Tpo3.PRE := 3000, [97].Timer.Tpo4.PRE := 10000, [97].Timer.Tpo5.PRE := 3000, [97].Timer.Tpo6.PRE := 3000, [98].Timer.Tpo1.PRE := 5000, [98].Timer.Tpo2.PRE := 5000, [98].Timer.Tpo3.PRE := 3000, [98].Timer.Tpo4.PRE := 10000, [98].Timer.Tpo5.PRE := 3000, [98].Timer.Tpo6.PRE := 15000, [99].Timer.Tpo1.PRE := 5000, [99].Timer.Tpo2.PRE := 5000, [99].Timer.Tpo3.PRE := 3000, [99].Timer.Tpo4.PRE := 10000, [99].Timer.Tpo5.PRE := 3000, [99].Timer.Tpo6.PRE := 3000, [100].Timer.Tpo1.PRE := 5000, [100].Timer.Tpo2.PRE := 5000, [100].Timer.Tpo3.PRE := 3000, [100].Timer.Tpo4.PRE := 10000, [100].Timer.Tpo5.PRE := 3000, [100].Timer.Tpo6.PRE := 3000, [100].S.Bits1 := 593, [100].S.Bits2 := 2600960, [100].S.Bits3 := 1073807361, [100].Next := 114, [100].Color := 2, [101].Timer.Tpo1.PRE := 5000, [101].Timer.Tpo2.PRE := 5000,
        [101].Timer.Tpo3.PRE := 3000, [101].Timer.Tpo4.PRE := 10000, [101].Timer.Tpo5.PRE := 3000, [101].Timer.Tpo6.PRE := 3000, [101].S.Bits1 := 593, [101].S.Bits2 := 2600960, [101].S.Bits3 := 1073807361, [101].Next := 114, [101].Color := 2, [102].Timer.Tpo1.PRE := 5000, [102].Timer.Tpo2.PRE := 5000, [102].Timer.Tpo3.PRE := 3000, [102].Timer.Tpo4.PRE := 10000, [102].Timer.Tpo5.PRE := 3000, [102].Timer.Tpo6.PRE := 3000, [102].S.Bits1 := 593, [102].S.Bits2 := 2600960, [102].S.Bits3 := 1073807361, [102].Next := 114, [102].Color := 2, [103].Timer.Tpo1.PRE := 5000, [103].Timer.Tpo2.PRE := 5000, [103].Timer.Tpo3.PRE := 3000, [103].Timer.Tpo4.PRE := 10000, [103].Timer.Tpo5.PRE := 3000, [103].Timer.Tpo6.PRE := 3000, [103].S.Bits1 := 593, [103].S.Bits2 := 2600960, [103].S.Bits3 := 1073807361, [103].Next := 116, [103].Color := 2, [104].Timer.Tpo1.PRE := 5000, [104].Timer.Tpo2.PRE := 5000, [104].Timer.Tpo3.PRE := 3000, [104].Timer.Tpo4.PRE := 10000, [104].Timer.Tpo5.PRE := 3000, [104].Timer.Tpo6.PRE := 3000, [104].S.Bits1 := 593, [104].S.Bits2 := 2600960, [104].S.Bits3 := 1073807361, [104].Next := 116, [104].Color := 2, [105].Timer.Tpo1.PRE := 5000, [105].Timer.Tpo2.PRE := 5000, [105].Timer.Tpo3.PRE := 3000, [105].Timer.Tpo5.PRE := 3000, [105].Timer.Tpo6.PRE := 3000, [105].S.Bits1 := 593, [105].S.Bits2 := 2600960, [105].S.Bits3 := 1073807361, [105].Next := 116, [105].Color := 2, [106].Timer.Tpo1.PRE := 5000, [106].Timer.Tpo2.PRE := 5000, [106].Timer.Tpo3.PRE := 3000, [106].Timer.Tpo5.PRE := 3000, [106].Timer.Tpo6.PRE := 3000, [107].Timer.Tpo1.PRE := 5000, [107].Timer.Tpo2.PRE := 5000, [107].Timer.Tpo3.PRE := 3000,
        [107].Timer.Tpo4.PRE := 10000, [107].Timer.Tpo5.PRE := 5000, [107].Timer.Tpo6.PRE := 3000, [108].Timer.Tpo1.PRE := 5000, [108].Timer.Tpo2.PRE := 5000, [108].Timer.Tpo3.PRE := 3000, [108].Timer.Tpo4.PRE := 10000, [108].Timer.Tpo5.PRE := 5000, [108].Timer.Tpo6.PRE := 3000, [109].Timer.Tpo1.PRE := 5000, [109].Timer.Tpo2.PRE := 5000, [109].Timer.Tpo3.PRE := 3000, [109].Timer.Tpo4.PRE := 10000, [109].Timer.Tpo5.PRE := 3000, [109].Timer.Tpo6.PRE := 3000, [110].Timer.Tpo1.PRE := 5000, [110].Timer.Tpo2.PRE := 5000, [110].Timer.Tpo3.PRE := 3000, [110].Timer.Tpo4.PRE := 10000, [110].Timer.Tpo5.PRE := 3000, [110].Timer.Tpo6.PRE := 15000, [110].S.Bits1 := 4, [110].S.Bits2 := 1409024, [110].S.Bits3 := 16, [111].Timer.Tpo1.PRE := 5000, [111].Timer.Tpo2.PRE := 5000, [111].Timer.Tpo3.PRE := 3000, [111].Timer.Tpo4.PRE := 10000, [111].Timer.Tpo5.PRE := 3000, [111].Timer.Tpo6.PRE := 3000, [111].S.Bits1 := 593, [111].S.Bits2 := 495616, [111].S.Bits3 := 1073807360, [111].Next := 119, [111].Color := 2, [112].Timer.Tpo1.PRE := 5000, [112].Timer.Tpo2.PRE := 5000, [112].Timer.Tpo3.PRE := 3000, [112].Timer.Tpo4.PRE := 10000, [112].Timer.Tpo5.PRE := 3000, [112].Timer.Tpo6.PRE := 3000, [112].S.Bits1 := 4, [112].S.Bits2 := 1409024, [112].S.Bits3 := 16, [113].Timer.Tpo1.PRE := 5000, [113].Timer.Tpo2.PRE := 5000, [113].Timer.Tpo3.PRE := 3000, [113].Timer.Tpo4.PRE := 10000, [113].Timer.Tpo5.PRE := 3000, [113].Timer.Tpo6.PRE := 3000, [113].S.Bits1 := 593, [113].S.Bits2 := 495616, [113].S.Bits3 := 1073807360, [113].Next := 118, [113].Color := 2, [114].Timer.Tpo1.PRE := 5000, [114].Timer.Tpo2.PRE := 5000, [114].Timer.Tpo3.PRE := 3000, [114].Timer.Tpo4.PRE := 10000, [114].Timer.Tpo5.PRE := 3000,
        [114].Timer.Tpo6.PRE := 3000, [114].S.Bits1 := 4, [114].S.Bits2 := 1409024, [114].S.Bits3 := 16, [115].Timer.Tpo1.PRE := 5000, [115].Timer.Tpo2.PRE := 5000, [115].Timer.Tpo3.PRE := 3000, [115].Timer.Tpo4.PRE := 10000, [115].Timer.Tpo5.PRE := 3000, [115].Timer.Tpo6.PRE := 3000, [115].S.Bits1 := 593, [115].S.Bits2 := 495616, [115].S.Bits3 := 1073807360, [115].Next := 119, [115].Color := 2, [116].Timer.Tpo1.PRE := 5000, [116].Timer.Tpo2.PRE := 5000, [116].Timer.Tpo3.PRE := 3000, [116].Timer.Tpo4.PRE := 10000, [116].Timer.Tpo5.PRE := 3000, [116].Timer.Tpo6.PRE := 3000, [116].S.Bits1 := 4, [116].S.Bits2 := 1409024, [116].S.Bits3 := 16, [117].Timer.Tpo1.PRE := 5000, [117].Timer.Tpo2.PRE := 5000, [117].Timer.Tpo3.PRE := 3000, [117].Timer.Tpo5.PRE := 3000, [117].Timer.Tpo6.PRE := 15000, [117].S.Bits1 := 593, [117].S.Bits2 := 495616, [117].S.Bits3 := 1073807360, [117].Next := 119, [117].Color := 2, [118].Timer.Tpo1.PRE := 5000, [118].Timer.Tpo2.PRE := 5000, [118].Timer.Tpo3.PRE := 3000, [118].Timer.Tpo5.PRE := 3000, [118].Timer.Tpo6.PRE := 15000, [118].S.Bits1 := 593, [118].S.Bits2 := 2600960, [118].S.Bits3 := 1073807361, [118].Next := 129, [118].Color := 2, [119].Timer.Tpo1.PRE := 5000, [119].Timer.Tpo2.PRE := 5000, [119].Timer.Tpo3.PRE := 3000, [119].Timer.Tpo4.PRE := 10000, [119].Timer.Tpo5.PRE := 5000, [119].Timer.Tpo6.PRE := 3000, [119].S.Bits1 := 593, [119].S.Bits2 := 2600960, [119].S.Bits3 := 1073807361, [119].Next := 129, [119].Color := 2, [120].Timer.Tpo1.PRE := 5000, [120].Timer.Tpo2.PRE := 5000, [120].Timer.Tpo3.PRE := 3000, [120].Timer.Tpo4.PRE := 10000, [120].Timer.Tpo5.PRE := 5000,
        [120].Timer.Tpo6.PRE := 3000, [120].S.Bits1 := 4, [120].S.Bits2 := 1409024, [120].S.Bits3 := 16, [121].Timer.Tpo1.PRE := 5000, [121].Timer.Tpo2.PRE := 5000, [121].Timer.Tpo3.PRE := 3000, [121].Timer.Tpo4.PRE := 10000, [121].Timer.Tpo5.PRE := 3000, [121].Timer.Tpo6.PRE := 3000, [121].S.Bits1 := 593, [121].S.Bits2 := 2600960, [121].S.Bits3 := 1073807361, [121].Next := 129, [121].Color := 2, [122].Timer.Tpo1.PRE := 5000, [122].Timer.Tpo2.PRE := 5000, [122].Timer.Tpo3.PRE := 3000, [122].Timer.Tpo4.PRE := 10000, [122].Timer.Tpo5.PRE := 3000, [122].Timer.Tpo6.PRE := 15000, [123].Timer.Tpo1.PRE := 5000, [123].Timer.Tpo2.PRE := 5000, [123].Timer.Tpo3.PRE := 3000, [123].Timer.Tpo4.PRE := 10000, [123].Timer.Tpo5.PRE := 3000, [123].Timer.Tpo6.PRE := 3000, [123].S.Bits1 := 65, [123].S.Bits2 := 495616, [123].S.Bits3 := 1073807360, [123].Next := 121, [123].Color := 2, [124].Timer.Tpo1.PRE := 5000, [124].Timer.Tpo2.PRE := 5000, [124].Timer.Tpo3.PRE := 3000, [124].Timer.Tpo4.PRE := 10000, [124].Timer.Tpo5.PRE := 3000, [124].Timer.Tpo6.PRE := 3000, [125].Timer.Tpo1.PRE := 5000, [125].Timer.Tpo2.PRE := 5000, [125].Timer.Tpo3.PRE := 3000, [125].Timer.Tpo4.PRE := 10000, [125].Timer.Tpo5.PRE := 3000, [125].Timer.Tpo6.PRE := 3000, [126].Timer.Tpo1.PRE := 5000, [126].Timer.Tpo2.PRE := 5000, [126].Timer.Tpo3.PRE := 3000, [126].Timer.Tpo4.PRE := 10000, [126].Timer.Tpo5.PRE := 3000, [126].Timer.Tpo6.PRE := 3000, [127].Timer.Tpo1.PRE := 5000, [127].Timer.Tpo2.PRE := 5000, [127].Timer.Tpo3.PRE := 3000, [127].Timer.Tpo4.PRE := 10000, [127].Timer.Tpo5.PRE := 3000, [127].Timer.Tpo6.PRE := 3000, [128].Timer.Tpo1.PRE := 5000, [128].Timer.Tpo2.PRE := 5000, [128].Timer.Tpo3.PRE := 3000, [128].Timer.Tpo4.PRE := 10000,
        [128].Timer.Tpo5.PRE := 3000, [128].Timer.Tpo6.PRE := 3000, [129].Timer.Tpo1.PRE := 5000, [129].Timer.Tpo2.PRE := 5000, [129].Timer.Tpo3.PRE := 3000, [129].Timer.Tpo4.PRE := 10000, [129].Timer.Tpo5.PRE := 3000, [129].Timer.Tpo6.PRE := 3000, [129].S.Bits1 := 4, [129].S.Bits2 := 1409024, [129].S.Bits3 := 16, [130].Timer.Tpo1.PRE := 5000, [130].Timer.Tpo2.PRE := 5000, [130].Timer.Tpo3.PRE := 3000, [130].Timer.Tpo4.PRE := 10000, [130].Timer.Tpo5.PRE := 3000, [130].Timer.Tpo5.ACC := 3190, [130].Timer.Tpo5.EN := 1, [130].Timer.Tpo5.DN := 1, [130].Timer.Tpo6.PRE := 3000, [130].S.Bits1 := 29, [130].S.Bits2 := -2010664959, [130].S.Bits3 := 1073807377, [130].Next := 129, [131].Timer.Tpo1.PRE := 5000, [131].Timer.Tpo2.PRE := 5000, [131].Timer.Tpo3.PRE := 3000, [131].Timer.Tpo4.PRE := 10000, [131].Timer.Tpo5.PRE := 3000, [131].Timer.Tpo6.PRE := 3000, [131].S.Bits1 := 593, [131].S.Bits2 := 2600960, [131].S.Bits3 := 1073807361, [131].Next := 132, [131].Color := 2, [132].Timer.Tpo1.PRE := 5000, [132].Timer.Tpo2.PRE := 5000, [132].Timer.Tpo3.PRE := 3000, [132].Timer.Tpo4.PRE := 10000, [132].Timer.Tpo5.PRE := 3000, [132].Timer.Tpo6.PRE := 3000, [132].S.Bits1 := 4, [132].S.Bits2 := 1409024, [132].S.Bits3 := 16, [133].Timer.Tpo1.PRE := 5000, [133].Timer.Tpo2.PRE := 5000, [133].Timer.Tpo3.PRE := 3000, [133].Timer.Tpo4.PRE := 10000, [133].Timer.Tpo4.EN := 1, [133].Timer.Tpo4.DN := 1, [133].Timer.Tpo5.PRE := 3000, [133].Timer.Tpo5.ACC := 3198, [133].Timer.Tpo5.EN := 1, [133].Timer.Tpo5.DN := 1, [133].Timer.Tpo6.PRE := 3000, [133].S.Bits1 := 221, [133].S.Bits2 := -1993887743, [133].S.Bits3 := -2147413999, [133].Next := 134, [133].Color := 6,
        [134].Timer.Tpo1.PRE := 5000, [134].Timer.Tpo2.PRE := 5000, [134].Timer.Tpo3.PRE := 3000, [134].Timer.Tpo4.PRE := 10000, [134].Timer.Tpo4.EN := 1, [134].Timer.Tpo4.DN := 1, [134].Timer.Tpo5.PRE := 3000, [134].Timer.Tpo5.ACC := 3191, [134].Timer.Tpo5.EN := 1, [134].Timer.Tpo5.DN := 1, [134].Timer.Tpo6.PRE := 3000, [134].S.Bits1 := 221, [134].S.Bits2 := -1993887743, [134].S.Bits3 := -2147413743, [134].Next := 137, [134].Color := 6, [135].Timer.Tpo1.PRE := 5000, [135].Timer.Tpo2.PRE := 5000, [135].Timer.Tpo3.PRE := 3000, [135].Timer.Tpo4.PRE := 10000, [135].Timer.Tpo5.PRE := 3000, [135].Timer.Tpo6.PRE := 3000, [135].S.Bits1 := 1, [135].S.Bits2 := 134713344, [136].Timer.Tpo1.PRE := 5000, [136].Timer.Tpo2.PRE := 5000, [136].Timer.Tpo3.PRE := 3000, [136].Timer.Tpo4.PRE := 10000, [136].Timer.Tpo5.PRE := 3000, [136].Timer.Tpo6.PRE := 3000, [136].S.Bits1 := 1, [136].S.Bits2 := 495616, [137].Timer.Tpo1.PRE := 5000, [137].Timer.Tpo2.PRE := 5000, [137].Timer.Tpo3.PRE := 3000, [137].Timer.Tpo4.PRE := 10000, [137].Timer.Tpo4.EN := 1, [137].Timer.Tpo4.DN := 1, [137].Timer.Tpo5.PRE := 3000, [137].Timer.Tpo5.ACC := 3210, [137].Timer.Tpo5.EN := 1, [137].Timer.Tpo5.DN := 1, [137].Timer.Tpo6.PRE := 3000, [137].S.Bits1 := 221, [137].S.Bits2 := -1993887743, [137].S.Bits3 := -2147413743, [137].Next := 171, [137].Color := 6, [138].Timer.Tpo1.PRE := 5000, [138].Timer.Tpo2.PRE := 5000, [138].Timer.Tpo3.PRE := 3000, [138].Timer.Tpo4.PRE := 10000, [138].Timer.Tpo5.PRE := 3000, [138].Timer.Tpo6.PRE := 3000, [138].S.Bits1 := 1041, [138].S.Bits2 := 136810501, [139].Timer.Tpo1.PRE := 5000, [139].Timer.Tpo2.PRE := 5000, [139].Timer.Tpo3.PRE := 3000, [139].Timer.Tpo4.PRE := 10000,
        [139].Timer.Tpo5.PRE := 3000, [139].Timer.Tpo6.PRE := 3000, [140].Timer.Tpo1.PRE := 5000, [140].Timer.Tpo2.PRE := 5000, [140].Timer.Tpo3.PRE := 3000, [140].Timer.Tpo4.PRE := 10000, [140].Timer.Tpo5.PRE := 3000, [140].Timer.Tpo6.PRE := 3000, [140].S.Bits1 := 4, [140].S.Bits2 := 1409024, [140].S.Bits3 := 16, [141].Timer.Tpo1.PRE := 5000, [141].Timer.Tpo2.PRE := 5000, [141].Timer.Tpo3.PRE := 3000, [141].Timer.Tpo4.PRE := 10000, [141].Timer.Tpo5.PRE := 3000, [141].Timer.Tpo6.PRE := 3000, [141].S.Bits1 := 593, [141].S.Bits2 := 2600960, [141].S.Bits3 := 1073807361, [141].Next := 152, [141].Color := 2, [142].Timer.Tpo1.PRE := 5000, [142].Timer.Tpo2.PRE := 5000, [142].Timer.Tpo3.PRE := 3000, [142].Timer.Tpo4.PRE := 10000, [142].Timer.Tpo5.PRE := 3000, [142].Timer.Tpo6.PRE := 3000, [143].Timer.Tpo1.PRE := 5000, [143].Timer.Tpo2.PRE := 5000, [143].Timer.Tpo3.PRE := 3000, [143].Timer.Tpo4.PRE := 10000, [143].Timer.Tpo5.PRE := 3000, [143].Timer.Tpo6.PRE := 3000, [144].Timer.Tpo1.PRE := 5000, [144].Timer.Tpo2.PRE := 5000, [144].Timer.Tpo3.PRE := 3000, [144].Timer.Tpo4.PRE := 10000, [144].Timer.Tpo5.PRE := 3000, [144].Timer.Tpo6.PRE := 3000, [145].Timer.Tpo1.PRE := 5000, [145].Timer.Tpo2.PRE := 5000, [145].Timer.Tpo3.PRE := 3000, [145].Timer.Tpo4.PRE := 10000, [145].Timer.Tpo5.PRE := 3000, [145].Timer.Tpo6.PRE := 3000, [146].Timer.Tpo1.PRE := 5000, [146].Timer.Tpo2.PRE := 5000, [146].Timer.Tpo3.PRE := 3000, [146].Timer.Tpo4.PRE := 10000, [146].Timer.Tpo5.PRE := 3000, [146].Timer.Tpo6.PRE := 3000, [147].Timer.Tpo1.PRE := 5000, [147].Timer.Tpo2.PRE := 5000, [147].Timer.Tpo3.PRE := 3000, [147].Timer.Tpo4.PRE := 10000, [147].Timer.Tpo5.PRE := 3000, [147].Timer.Tpo6.PRE := 3000, [148].Timer.Tpo1.PRE := 5000, [148].Timer.Tpo2.PRE := 5000,
        [148].Timer.Tpo3.PRE := 3000, [148].Timer.Tpo4.PRE := 10000, [148].Timer.Tpo5.PRE := 3000, [148].Timer.Tpo6.PRE := 3000, [149].Timer.Tpo1.PRE := 5000, [149].Timer.Tpo2.PRE := 5000, [149].Timer.Tpo3.PRE := 3000, [149].Timer.Tpo4.PRE := 10000, [149].Timer.Tpo5.PRE := 3000, [149].Timer.Tpo6.PRE := 3000, [150].Timer.Tpo1.PRE := 5000, [150].Timer.Tpo2.PRE := 5000, [150].Timer.Tpo3.PRE := 3000, [150].Timer.Tpo4.PRE := 10000, [150].Timer.Tpo5.PRE := 3000, [150].Timer.Tpo6.PRE := 3000, [150].S.Bits1 := 4, [150].S.Bits2 := 1409024, [150].S.Bits3 := 16, [151].Timer.Tpo1.PRE := 5000, [151].Timer.Tpo2.PRE := 5000, [151].Timer.Tpo3.PRE := 3000, [151].Timer.Tpo4.PRE := 10000, [151].Timer.Tpo5.PRE := 3000, [151].Timer.Tpo6.PRE := 3000, [151].S.Bits1 := 593, [151].S.Bits2 := 2600960, [151].S.Bits3 := 1073807361, [151].Next := 152, [151].Color := 2, [152].Timer.Tpo1.PRE := 5000, [152].Timer.Tpo2.PRE := 5000, [152].Timer.Tpo3.PRE := 3000, [152].Timer.Tpo4.PRE := 10000, [152].Timer.Tpo5.PRE := 3000, [152].Timer.Tpo6.PRE := 3000, [152].S.Bits1 := 4, [152].S.Bits2 := 1409024, [152].S.Bits3 := 16, [153].Timer.Tpo1.PRE := 5000, [153].Timer.Tpo2.PRE := 5000, [153].Timer.Tpo3.PRE := 3000, [153].Timer.Tpo4.PRE := 10000, [153].Timer.Tpo5.PRE := 3000, [153].Timer.Tpo6.PRE := 3000, [153].S.Bits1 := 593, [153].S.Bits2 := 2600960, [153].S.Bits3 := 1073807361, [153].Next := 20, [153].Color := 2, [154].Timer.Tpo1.PRE := 5000, [154].Timer.Tpo2.PRE := 5000, [154].Timer.Tpo3.PRE := 3000, [154].Timer.Tpo4.PRE := 10000, [154].Timer.Tpo5.PRE := 3000, [154].Timer.Tpo6.PRE := 3000, [154].S.Bits1 := 593, [154].S.Bits2 := 2600960, [154].S.Bits3 := 1073807361, [154].Next := 21,
        [154].Color := 2, [155].Timer.Tpo1.PRE := 5000, [155].Timer.Tpo2.PRE := 5000, [155].Timer.Tpo3.PRE := 3000, [155].Timer.Tpo4.PRE := 10000, [155].Timer.Tpo5.PRE := 3000, [155].Timer.Tpo6.PRE := 3000, [155].S.Bits1 := 593, [155].S.Bits2 := 2600960, [155].S.Bits3 := 1073807361, [155].Next := 22, [155].Color := 2, [156].Timer.Tpo1.PRE := 5000, [156].Timer.Tpo2.PRE := 5000, [156].Timer.Tpo3.PRE := 3000, [156].Timer.Tpo4.PRE := 10000, [156].Timer.Tpo5.PRE := 3000, [156].Timer.Tpo6.PRE := 3000, [156].S.Bits1 := 593, [156].S.Bits2 := 2600960, [156].S.Bits3 := 1073807361, [156].Next := 23, [156].Color := 2, [157].Timer.Tpo1.PRE := 5000, [157].Timer.Tpo2.PRE := 5000, [157].Timer.Tpo3.PRE := 3000, [157].Timer.Tpo4.PRE := 10000, [157].Timer.Tpo5.PRE := 3000, [157].Timer.Tpo6.PRE := 3000, [157].S.Bits1 := 593, [157].S.Bits2 := 2600960, [157].S.Bits3 := 1073807361, [157].Next := 24, [157].Color := 2, [158].Timer.Tpo1.PRE := 5000, [158].Timer.Tpo2.PRE := 5000, [158].Timer.Tpo3.PRE := 3000, [158].Timer.Tpo4.PRE := 10000, [158].Timer.Tpo5.PRE := 3000, [158].Timer.Tpo6.PRE := 3000, [158].S.Bits1 := 593, [158].S.Bits2 := 2600960, [158].S.Bits3 := 1073807361, [158].Next := 25, [158].Color := 2, [159].Timer.Tpo1.PRE := 5000, [159].Timer.Tpo2.PRE := 5000, [159].Timer.Tpo3.PRE := 3000, [159].Timer.Tpo4.PRE := 10000, [159].Timer.Tpo5.PRE := 3000, [159].Timer.Tpo6.PRE := 3000, [159].S.Bits1 := 593, [159].S.Bits2 := 2600960, [159].S.Bits3 := 1073807361, [159].Next := 26, [159].Color := 2, [160].Timer.Tpo1.PRE := 5000, [160].Timer.Tpo2.PRE := 5000, [160].Timer.Tpo3.PRE := 3000, [160].Timer.Tpo4.PRE := 10000,
        [160].Timer.Tpo5.PRE := 3000, [160].Timer.Tpo6.PRE := 3000, [160].S.Bits1 := 593, [160].S.Bits2 := 2600960, [160].S.Bits3 := 1073807361, [160].Next := 27, [160].Color := 2, [161].Timer.Tpo1.PRE := 5000, [161].Timer.Tpo2.PRE := 5000, [161].Timer.Tpo3.PRE := 3000, [161].Timer.Tpo4.PRE := 10000, [161].Timer.Tpo5.PRE := 3000, [161].Timer.Tpo6.PRE := 3000, [161].S.Bits1 := 593, [161].S.Bits2 := 2600960, [161].S.Bits3 := 1073807361, [161].Next := 28, [161].Color := 2, [162].Timer.Tpo1.PRE := 5000, [162].Timer.Tpo2.PRE := 5000, [162].Timer.Tpo3.PRE := 3000, [162].Timer.Tpo4.PRE := 10000, [162].Timer.Tpo5.PRE := 3000, [162].Timer.Tpo6.PRE := 3000, [162].S.Bits1 := 593, [162].S.Bits2 := 2600960, [162].S.Bits3 := 1073807361, [162].Next := 29, [162].Color := 2, [163].Timer.Tpo1.PRE := 5000, [163].Timer.Tpo2.PRE := 5000, [163].Timer.Tpo3.PRE := 3000, [163].Timer.Tpo4.PRE := 10000, [163].Timer.Tpo5.PRE := 3000, [163].Timer.Tpo6.PRE := 3000, [163].S.Bits1 := 593, [163].S.Bits2 := 2600960, [163].S.Bits3 := 1073807361, [163].Next := 30, [163].Color := 2, [164].Timer.Tpo1.PRE := 5000, [164].Timer.Tpo2.PRE := 5000, [164].Timer.Tpo3.PRE := 3000, [164].Timer.Tpo4.PRE := 10000, [164].Timer.Tpo5.PRE := 3000, [164].Timer.Tpo6.PRE := 3000, [164].S.Bits1 := 593, [164].S.Bits2 := 2600960, [164].S.Bits3 := 1073807361, [164].Next := 31, [164].Color := 2, [165].Timer.Tpo1.PRE := 5000, [165].Timer.Tpo2.PRE := 5000, [165].Timer.Tpo3.PRE := 3000, [165].Timer.Tpo4.PRE := 10000, [165].Timer.Tpo5.PRE := 3000, [165].Timer.Tpo6.PRE := 3000, [165].S.Bits1 := 593, [165].S.Bits2 := 2600960, [165].S.Bits3 := 1073807361,
        [165].Next := 32, [165].Color := 2, [166].Timer.Tpo1.PRE := 5000, [166].Timer.Tpo2.PRE := 5000, [166].Timer.Tpo3.PRE := 3000, [166].Timer.Tpo4.PRE := 10000, [166].Timer.Tpo5.PRE := 3000, [166].Timer.Tpo6.PRE := 3000, [166].S.Bits1 := 593, [166].S.Bits2 := 2600960, [166].S.Bits3 := 1073807361, [166].Next := 33, [166].Color := 2, [167].Timer.Tpo1.PRE := 5000, [167].Timer.Tpo2.PRE := 5000, [167].Timer.Tpo3.PRE := 3000, [167].Timer.Tpo4.PRE := 10000, [167].Timer.Tpo5.PRE := 3000, [167].Timer.Tpo6.PRE := 3000, [167].S.Bits1 := 593, [167].S.Bits2 := 2600960, [167].S.Bits3 := 1073807361, [167].Next := 34, [167].Color := 2, [168].Timer.Tpo1.PRE := 5000, [168].Timer.Tpo2.PRE := 5000, [168].Timer.Tpo3.PRE := 3000, [168].Timer.Tpo4.PRE := 10000, [168].Timer.Tpo5.PRE := 3000, [168].Timer.Tpo6.PRE := 3000, [168].S.Bits1 := 593, [168].S.Bits2 := 2600960, [168].S.Bits3 := 1073807361, [168].Next := 35, [168].Color := 2, [169].Timer.Tpo1.PRE := 5000, [169].Timer.Tpo2.PRE := 5000, [169].Timer.Tpo3.PRE := 3000, [169].Timer.Tpo4.PRE := 10000, [169].Timer.Tpo5.PRE := 3000, [169].Timer.Tpo6.PRE := 3000, [170].Timer.Tpo1.PRE := 5000, [170].Timer.Tpo2.PRE := 5000, [170].Timer.Tpo3.PRE := 3000, [170].Timer.Tpo4.PRE := 10000, [170].Timer.Tpo5.PRE := 3000, [170].Timer.Tpo6.PRE := 3000, [170].S.Bits1 := 224, [170].S.Bits2 := 1146880, [170].Next := 26, [170].Color := 7, [171].Timer.Tpo1.PRE := 5000, [171].Timer.Tpo2.PRE := 5000, [171].Timer.Tpo3.PRE := 3000, [171].Timer.Tpo4.PRE := 10000, [171].Timer.Tpo5.PRE := 3000, [171].Timer.Tpo6.PRE := 3000, [171].S.Bits1 := 68, [171].S.Bits2 := 1146880, [171].S.Bits3 := 256,
        [171].Next := 150, [171].Color := 2, [172].Timer.Tpo1.PRE := 5000, [172].Timer.Tpo2.PRE := 5000, [172].Timer.Tpo3.PRE := 3000, [172].Timer.Tpo4.PRE := 10000, [172].Timer.Tpo5.PRE := 3000, [172].Timer.Tpo6.PRE := 3000, [173].Timer.Tpo1.PRE := 5000, [173].Timer.Tpo2.PRE := 5000, [173].Timer.Tpo3.PRE := 3000, [173].Timer.Tpo4.PRE := 10000, [173].Timer.Tpo5.PRE := 3000, [173].Timer.Tpo6.PRE := 3000, [174].Timer.Tpo1.PRE := 5000, [174].Timer.Tpo2.PRE := 5000, [174].Timer.Tpo3.PRE := 3000, [174].Timer.Tpo4.PRE := 10000, [174].Timer.Tpo5.PRE := 3000, [174].Timer.Tpo6.PRE := 3000, [175].Timer.Tpo1.PRE := 5000, [175].Timer.Tpo2.PRE := 5000, [175].Timer.Tpo3.PRE := 3000, [175].Timer.Tpo4.PRE := 10000, [175].Timer.Tpo5.PRE := 3000, [175].Timer.Tpo6.PRE := 3000, [176].Timer.Tpo1.PRE := 5000, [176].Timer.Tpo2.PRE := 5000, [176].Timer.Tpo3.PRE := 3000, [176].Timer.Tpo4.PRE := 10000, [176].Timer.Tpo5.PRE := 3000, [176].Timer.Tpo6.PRE := 3000, [177].Timer.Tpo1.PRE := 5000, [177].Timer.Tpo2.PRE := 5000, [177].Timer.Tpo3.PRE := 3000, [177].Timer.Tpo4.PRE := 10000, [177].Timer.Tpo5.PRE := 3000, [177].Timer.Tpo6.PRE := 3000, [178].Timer.Tpo1.PRE := 5000, [178].Timer.Tpo2.PRE := 5000, [178].Timer.Tpo3.PRE := 3000, [178].Timer.Tpo4.PRE := 10000, [178].Timer.Tpo5.PRE := 3000, [178].Timer.Tpo6.PRE := 3000, [179].Timer.Tpo1.PRE := 5000, [179].Timer.Tpo2.PRE := 5000, [179].Timer.Tpo3.PRE := 3000, [179].Timer.Tpo4.PRE := 10000, [179].Timer.Tpo5.PRE := 3000, [179].Timer.Tpo6.PRE := 3000, [180].Timer.Tpo1.PRE := 5000, [180].Timer.Tpo2.PRE := 5000, [180].Timer.Tpo3.PRE := 3000, [180].Timer.Tpo4.PRE := 10000, [180].Timer.Tpo5.PRE := 3000, [180].Timer.Tpo6.PRE := 3000, [200].S.Bits2 := 1146880, [201].S.Bits2 := 1146880, [202].S.Bits2 := 1146880, [203].S.Bits2 := 1146880,
        [204].S.Bits2 := 1146880, [205].S.Bits2 := 1146880, [206].S.Bits2 := 1146880, [207].S.Bits2 := 1146880, [208].S.Bits2 := 1146880, [209].S.Bits2 := 1146880, [210].S.Bits2 := 1146880, [211].S.Bits2 := 1146880, [212].S.Bits2 := 1146880, [213].S.Bits2 := 1146880, [214].S.Bits2 := 1146880, [215].S.Bits2 := 1146880, [216].S.Bits2 := 1146880, [217].S.Bits2 := 1146880, [218].S.Bits2 := 1146880, [219].S.Bits2 := 1146880, [220].S.Bits2 := 1146880, [221].S.Bits2 := 1146880, [222].S.Bits2 := 1146880, [223].S.Bits2 := 1146880, [224].S.Bits2 := 1146880, [225].S.Bits2 := 1146880, [226].S.Bits2 := 1146880, [227].S.Bits2 := 1146880, [228].S.Bits2 := 1146880, [229].S.Bits2 := 1146880, [230].S.Bits2 := 1146880, [231].S.Bits2 := 1146880, [232].S.Bits2 := 1146880, [233].S.Bits2 := 1146880, [234].S.Bits2 := 1146880, [235].S.Bits2 := 1146880, [236].S.Bits2 := 1146880, [237].S.Bits2 := 1146880, [238].S.Bits2 := 1146880, [239].S.Bits2 := 1146880, [240].S.Bits2 := 1146880, [241].S.Bits2 := 1146880, [242].S.Bits2 := 1146880, [243].S.Bits2 := 1146880, [244].S.Bits2 := 1146880, [245].S.Bits2 := 1146880, [246].S.Bits2 := 1146880, [247].S.Bits2 := 1146880, [248].S.Bits2 := 1146880, [249].S.Bits2 := 1146880, [250].S.Bits2 := 1146880, [251].S.Bits2 := 1146880, [252].S.Bits2 := 1146880, [253].S.Bits2 := 1146880, [254].S.Bits2 := 1146880, [255].S.Bits2 := 1146880, [256].S.Bits2 := 1146880, [257].S.Bits2 := 1146880, [258].S.Bits2 := 1146880, [259].S.Bits2 := 1146880, [260].S.Bits2 := 1146880, [261].S.Bits2 := 1146880, [262].S.Bits2 := 1146880, [263].S.Bits2 := 1146880,
        [264].S.Bits2 := 1146880, [265].S.Bits2 := 1146880, [266].S.Bits2 := 1146880, [267].S.Bits2 := 1146880, [268].S.Bits2 := 1146880, [269].S.Bits2 := 1146880, [270].S.Bits2 := 1146880, [271].S.Bits2 := 1146880, [272].S.Bits2 := 1146880, [273].S.Bits2 := 1146880, [274].S.Bits2 := 1146880, [275].S.Bits2 := 1146880, [276].S.Bits2 := 1146880, [277].S.Bits2 := 1146880, [278].S.Bits2 := 1146880, [279].S.Bits2 := 1146880, [280].S.Bits2 := 1146880, [281].S.Bits2 := 1146880, [282].S.Bits2 := 1146880, [283].S.Bits2 := 1146880, [284].S.Bits2 := 1146880, [285].S.Bits2 := 1146880, [286].S.Bits2 := 1146880, [287].S.Bits2 := 1146880, [288].S.Bits2 := 1146880, [289].S.Bits2 := 1146880, [290].S.Bits2 := 1146880, [291].S.Bits2 := 1146880, [292].S.Bits2 := 1146880, [293].S.Bits2 := 1146880, [294].S.Bits2 := 1146880, [295].S.Bits2 := 1146880, [296].S.Bits2 := 1146880, [297].S.Bits2 := 1146880, [298].S.Bits2 := 1146880, [299].S.Bits2 := 1146880, [300].S.Bits2 := 1146880);
        [4].S.BITS1.30   // 7-RED-1004 Falla Partida
        [5].S.BITS1.2   // 7-RED-1005 Conf. Marcha
        [6].S.BITS1.2   // 7-COM-1006 Conf Pos Abrir
        [7].S.BITS1.2   // 7-COM-1007 Conf Pos Abrir
        [7].S.BITS2.7   // MAG-604-01 Disable Codes
        [8].S.BITS1.2   // 7-COM-1008 Conf Pos Abrir
        [8].S.BITS2.7   // MAG-604-02 Disable Codes
        [9].S.BITS1.2   // 7-COM-1009 Conf Pos Abrir
        [9].S.BITS2.7   // MAG-604-03 Disable Codes
        [13].S.BITS1.1   // 7-CON-1013 Falla Resumen
        [14].S.BITS1.9   // 90-CAN-001 Conf. Cerrado
        [14].S.BITS1.1   // 7-CON-1014 Falla Resumen
        [14].S.BITS1.30   // 7-CON-1014 Falla Cerrar
        [16].S.BITS1.1   // 7-LMG-1016 Falla Resumen
        [17].S.BITS1.1   // 7-ELV-1017 Falla Resumen
        [1].S.BITS1.8   // CV-11_LL
        [18].S.BITS1.1   // 7-BIF-1018 Falla Resumen
        [15].S.BITS1.9   // 90-CAN-002 Conf. Cerrado
        [1].S.BITS1.9   // CV-11LM
        [1].S.BITS1.10   // CV-11LH
        [1].S.BITS1.29   // CV-11 Falla Abrir
        [1].S.BITS2.11   // VOL-600-00 Enc Ext
        [26].S.BITS1.1   // 7-CON-1026 Falla Resumen
        [27].S.BITS1.1   // 7-BIF-1027 Falla Resumen
        [32].S.BITS1.1   // 7-RED-1053 Falla Resumen
        [1].S.BITS2.31   // CV-11 OUT OPEN
        [33].S.BITS1.1   // 7-CON-1054 Falla Resumen
        [34].S.BITS1.1   // 7-BIF-1055 Falla Resumen
        [2].S.BITS1.8   // CV-12LL
        [2].S.BITS1.9   // CV-12LM
        [2].S.BITS1.10   // CV-12LH
        [35].S.BITS1.1   // 7-CON-1055 Falla Resumen
        [2].S.BITS1.29   // CV-12 Falla Abrir
        [35].S.BITS1.30   // 7-CON-1055 Falla Cerrar
        [135].S.BITS1.27   // RIB-33 FV0
        [36].S.BITS1.1   // 60-VEN-002 Falla Resumen
        [37].S.BITS1.2   // 60-VEN-004A Conf. Marcha
        [37].S.BITS2.20   // 60-VEN-004A Reset Falla
        [2].S.BITS2.31   // CV-12 OUT OPEN
        [37].S.BITS2.27   // 60-VEN-004A Cmd. Marcha
        [3].S.BITS1.8   // RED-602-00 IAto
        [38].S.BITS1.30   // 60-TOR-002Falla Partida
        [39].S.BITS1.1   // 60-TOR-002 Falla Resumen
        [3].S.BITS1.10   // RED-602-00 IV0
        [40].S.BITS1.1   // 7-VRT-1064 Falla Resumen
        [3].S.BITS2.11   // RED-602-00 Enc Ext
        [42].S.BITS1.1   // 7-FLT-1066 Falla Resumen
        [43].S.BITS1.1   // 7-VEN-1067 Falla Resumen
        [4].S.BITS1.0   // 7-RED-1004 Enable
        [4].S.BITS1.1   // 7-RED-1004 Falla Resumen
        [4].S.BITS1.2   // 7-RED-1004 Conf. Marcha
        [44].S.BITS1.1   // 90-FIL-001 Falla Resumen
        [4].S.BITS1.8   // ELE-606-00 IAto
        [45].S.BITS1.1   // 7-ROS-1068 Falla Resumen
        [16].S.BITS1.9   // 90-CAN-003 Conf. Cerrado
        [46].S.BITS1.1   // 7-ROS-1069 Falla Resumen
        [47].S.BITS2.20   // 7-ELV-1070 Reset Falla
        [47].S.BITS2.27   // 7-ELV-1070 Cmd. Marcha
        [48].S.BITS1.9   // 60-MMA-001T LM
        [4].S.BITS1.10   // ELE-606-00 IV0
        [48].S.BITS1.26   // 7-RED-1071 FLL
        [4].S.BITS1.26   // 7-RED-1004 FLL
        [48].S.BITS1.27   // 7-RED-1071 FV0
        [4].S.BITS1.27   // 7-RED-1004 FV0
        [48].S.BITS1.28   // 7-RED-1071 FATO
        [4].S.BITS1.28   // 7-RED-1004 FATO
        [4].S.BITS2.11   // ELE-606-00 Enc Ext
        [4].S.BITS2.20   // 7-RED-1004 Reset Falla
        [4].S.BITS2.23   // 7-RED-1004 Test
        [4].S.BITS2.27   // 7-RED-1004 Cmd. Marcha
        [49].S.BITS1.0   // 7-CON-1072 Enable
        [4].S.BITS2.30   // 7-RED-1004 OUT MARCHA
        [49].S.BITS1.1   // 7-CON-1072 Falla Resumen
        [4].S.BITS2.31   // ELE-606-00 Out
        [60].S.BITS1.1   // CV-4 Falla Resumen
        [5].S.BITS1.0   // 7-RED-1005 Enable
        [49].S.BITS1.26   // 90-TOR-001 FLL
        [5].S.BITS1.1   // 7-RED-1005 Falla Resumen
        [49].S.BITS1.27   // 90-TOR-001 FV0
        [5].S.BITS1.8   // ZAR-607-00 IAto
        [49].S.BITS1.28   // 90-TOR-001 FATO
        [5].S.BITS1.29   // 60-CAN-005 Falla Abrir
        [49].S.BITS2.20   // 7-CON-1072 Reset Falla
        [49].S.BITS2.23   // 7-CON-1072 Test
        [5].S.BITS2.11   // ZAR-607-00 Enc Ext
        [49].S.BITS2.27   // 7-CON-1072 Cmd. Open
        [5].S.BITS2.20   // 7-RED-1005 Reset Falla
        [49].S.BITS2.30   // 7-CON-1072 OUT CLOSE
        [5].S.BITS2.23   // 7-RED-1005 Test
        [50].S.BITS1.0   // 7-CON-1073 Enable
        [50].S.BITS1.1   // 7-CON-1073 Falla Resumen
        [6].S.BITS1.0   // 7-COM-1006 Enable
        [60].S.BITS2.30   // CV-4 OUT CLOSE
        [6].S.BITS1.1   // 7-COM-1006 Falla Resumen
        [327].S.BITS2.31   // CV-9 OUT OPEN
        [6].S.BITS1.8   // MAG-604-00 IAto
        [50].S.BITS1.26   // 90-TAB-002 FLL
        [6].S.BITS1.29   // 7-COM-1006 Falla Abrir
        [50].S.BITS1.27   // 90-TAB-002 FV0
        [6].S.BITS1.30   // 7-COM-1006 Falla Cerrar
        [50].S.BITS1.28   // 90-TAB-002 FATO
        [6].S.BITS2.11   // MAG-604-00 Enc Ext
        [50].S.BITS2.11   // RED-657-00 Enc Ext
        [6].S.BITS2.20   // 7-COM-1006 Reset Falla
        [50].S.BITS2.20   // 7-CON-1073 Reset Falla
        [6].S.BITS2.23   // 7-COM-1006 Test
        [50].S.BITS2.23   // 7-CON-1073 Test
        [6].S.BITS2.27   // 7-COM-1006 Cmd. Open
        [50].S.BITS2.27   // 7-CON-1073 Cmd. Open
        [6].S.BITS2.30   // 7-COM-1006 OUT CLOSE
        [50].S.BITS2.30   // 7-CON-1073 OUT CLOSE
        [7].S.BITS1.0   // 7-COM-1007 Enable
        [7].S.BITS1.1   // 7-COM-1007 Falla Resumen
        [51].S.BITS1.0   // 7-CON-1074 Enable
        [7].S.BITS1.9   // MAG-604-01 IClose
        [51].S.BITS1.1   // 7-CON-1074 Falla Resumen
        [7].S.BITS1.10   // MAG-604-01 IOpen
        [51].S.BITS1.29   // 7-CON-1074 Falla Abrir
        [7].S.BITS1.29   // 7-COM-1007 Falla Abrir
        [51].S.BITS1.30   // 7-CON-1074 Falla Cerrar
        [77].S.BITS1.29   // 70-BIF-001 Falla Pos. Izquierda
        [7].S.BITS1.30   // 7-COM-1007 Falla Cerrar
        [51].S.BITS2.20   // 7-CON-1074 Reset Falla
        [7].S.BITS2.20   // 7-COM-1007 Reset Falla
        [51].S.BITS2.23   // 7-CON-1074 Test
        [7].S.BITS2.23   // 7-COM-1007 Test
        [51].S.BITS2.27   // 7-CON-1074 Cmd. Open
        [7].S.BITS2.27   // 7-COM-1007 Cmd. Open
        [52].S.BITS1.0   // 7-CON-1075 Enable
        [7].S.BITS2.30   // 7-COM-1007 OUT CLOSE
        [52].S.BITS1.1   // 7-CON-1075 Falla Resumen
        [7].S.BITS2.31   // 7-COM-1007 OUT OPEN
        [8].S.BITS1.0   // 7-COM-1008 Enable
        [8].S.BITS1.1   // 7-COM-1008 Falla Resumen
        [8].S.BITS1.29   // 7-COM-1008 Falla Abrir
        [8].S.BITS1.30   // 7-COM-1008 Falla Cerrar
        [8].S.BITS2.20   // 7-COM-1008 Reset Falla
        [77].S.BITS2.26   // 70-BIF-001 Cmd. Pos . Izquierda
        [101].S.BITS1.2   // 70-BIF-003 Conf. Pos. Izquierda
        [8].S.BITS2.23   // 7-COM-1008 Test
        [8].S.BITS2.27   // 7-COM-1008 Cmd. Open
        [8].S.BITS2.30   // 7-COM-1008 OUT CLOSE
        [77].S.BITS1.2   // 7-RED-1090 Conf. Marcha
        [9].S.BITS1.0   // 7-COM-1009 Enable
        [91].S.BITS2.20   // CV-6 Reset Falla
        [9].S.BITS1.1   // 7-COM-1009 Falla Resumen
        [91].S.BITS2.23   // CV-6 Test
        [9].S.BITS1.9   // MAG-604-03 Izq.
        [91].S.BITS2.27   // CV-6 Cmd. Open
        [9].S.BITS1.10   // MAG-604-03 Der.
        [9].S.BITS1.29   // 7-COM-1009 Falla Abrir
        [91].S.BITS2.30   // CV-6 OUT CLOSE
        [9].S.BITS1.30   // 7-COM-1009 Falla Cerrar
        [52].S.BITS1.26   // 60-ALI-002 FLL
        [9].S.BITS2.20   // 7-COM-1009 Reset Falla
        [52].S.BITS1.27   // 60-ALI-002 FV0
        [9].S.BITS2.23   // 7-COM-1009 Test
        [150].S.BITS1.9   // 70-BIN-006 LM
        [52].S.BITS1.28   // 60-ALI-002 FATO
        [52].S.BITS2.20   // 7-CON-1075 Reset Falla
        [52].S.BITS2.23   // 7-CON-1075 Test
        [9].S.BITS2.27   // 7-COM-1009 Cmd. Open
        [52].S.BITS2.27   // 7-CON-1075 Cmd. Open
        [53].S.BITS1.0   // 7-RED-1076 Enable
        [9].S.BITS2.30   // 7-COM-1009 OUT CLOSE
        [91].S.BITS2.31   // CV-6 OUT OPEN
        [9].S.BITS2.31   // 7-COM-1009 OUT OPEN
        [53].S.BITS1.26   // 7-RED-1076 FLL
        [10].S.BITS1.9   // BIF-698-00 Izq.
        [53].S.BITS1.27   // 7-RED-1076 FV0
        [10].S.BITS2.31   // BIF-698-00 Cmd Der
        [11].S.BITS1.9   // TOL-604-00 LM
        [11].S.BITS1.26   // 60-TDC-002 FLL
        [11].S.BITS1.27   // 60-TDC-002 FV0
        [11].S.BITS1.28   // 60-TDC-002 FATO
        [135].S.BITS1.28   // RIB-33 FATO
        [53].S.BITS1.28   // 7-RED-1076 FATO
        [53].S.BITS2.23   // 7-RED-1076 Test
        [63].S.BITS1.9   // 90-MRO-001-A Sobrecarga
        [17].S.BITS1.9   // 90-CAN-004 Conf. Cerrado
        [12].S.BITS2.11   // RED-603-00 Enc Ext
        [14].S.BITS1.10   // 90-CAN-001 Conf. Abierto
        [105].S.BITS2.7   // CON-622-00Cmd Open
        [60].S.BITS2.23   // CV-4 Test
        [135].S.BITS2.7   // CON-693-00 Disable Codes
        [64].S.BITS1.9   // 90-MRO-001-B Sobrecarga
        [179].S.BITS1.8   // TOL-064-00 LL
        [179].S.BITS1.9   // TOL-064-00 LM
        [13].S.BITS1.0   // 7-CON-1013 Enable
        [677].S.BITS1.10   // 120-BIN-029 LH
        [13].S.BITS1.29   // 7-CON-1013 Falla Abrir
        [65].S.BITS1.9   // 7-BIN-1084 LM
        [13].S.BITS1.9   // 90-TDC-001 Sobrecarga
        [13].S.BITS2.11   // ELE-605-00 Enc Ext
        [13].S.BITS2.20   // 7-CON-1013 Reset Falla
        [13].S.BITS2.23   // 7-CON-1013 Test
        [18].S.BITS1.9   // 90-TDC-002 Sobrecarga
        [54].S.BITS1.0   // 7-CON-1077 Enable
        [25].S.BITS2.23   // 7-CON-1025 Test
        [26].S.BITS1.9   // 90-VEN-005 Sobrecarga
        [28].S.BITS1.9   // 7-TOL-1049 LM
        [93].S.BITS1.0   // TCS-44_M Enable
        [150].S.BITS1.10   // 70-BIN-006 LH
        [93].S.BITS1.1   // TCS-44_M Falla Resumen
        [560].S.BITS2.31   // CV-11 OUT OPEN
        [679].S.BITS1.10   // 120-BIN-030 LH
        [29].S.BITS1.9   // 90-TDC-005 Sobrecarga
        [54].S.BITS1.26   // 90-ALI-002 FLL
        [54].S.BITS1.27   // 90-ALI-002 FV0
        [14].S.BITS1.0   // 7-CON-1014 Enable
        [54].S.BITS1.28   // 90-ALI-002 FATO
        [54].S.BITS2.7   // CON-671-01Cmd Open
        [14].S.BITS1.8   // RED-640-00 IAto
        [54].S.BITS2.23   // 7-CON-1077 Test
        [54].S.BITS2.30   // 7-CON-1077 OUT CLOSE
        [55].S.BITS1.0   // 7-RED-1078 Enable
        [14].S.BITS1.29   // 7-CON-1014 Falla Abrir
        [60].S.BITS1.30   // CV-4 Falla Cerrar
        [14].S.BITS2.11   // RED-640-00 Enc Ext
        [233].S.BITS2.23   // 7-LMG-1187 Test
        [14].S.BITS2.20   // 7-CON-1014 Reset Falla
        [55].S.BITS1.26   // 7-RED-1078 FLL
        [14].S.BITS2.23   // 7-CON-1014 Test
        [55].S.BITS1.27   // 7-RED-1078 FV0
        [14].S.BITS2.27   // 7-CON-1014 Cmd. Open
        [93].S.BITS1.2   // TCS-44_M Conf. Marcha
        [242].S.BITS1.8   // 100-TOR-021 Atollo
        [14].S.BITS2.30   // 7-CON-1014 OUT CLOSE
        [55].S.BITS1.28   // 7-RED-1078 FATO
        [14].S.BITS2.31   // 7-CON-1014 OUT OPEN
        [55].S.BITS2.23   // 7-RED-1078 Test
        [40].S.BITS1.9   // 90-TAB-001 Sobrecarga
        [234].S.BITS2.23   // 100-CAN-023 Test
        [235].S.BITS2.23   // 7-LRT-1189 Test
        [16].S.BITS1.0   // 7-LMG-1016 Enable
        [93].S.BITS1.4   // TCS-44_M Cmd. Automatico
        [16].S.BITS1.29   // 90-CAN-003 Falla Abrir
        [56].S.BITS1.0   // 7-CON-1079 Enable
        [16].S.BITS2.20   // 7-LMG-1016 Reset Falla
        [16].S.BITS2.23   // 7-LMG-1016 Test
        [56].S.BITS1.1   // 7-CON-1079 Falla Resumen
        [236].S.BITS2.23   // 100-CAN-025 Test
        [327].S.BITS1.29   // CV-9 Falla Abrir
        [56].S.BITS1.29   // 7-CON-1079 Falla Abrir
        [19].S.BITS1.9   // 90-CAN-006 Conf. Cerrado
        [56].S.BITS2.20   // 7-CON-1079 Reset Falla
        [56].S.BITS2.23   // 7-CON-1079 Test
        [43].S.BITS1.9   // 90-ALI-001 Sobrecarga
        [45].S.BITS1.9   // 90-VEN-001 Sobrecarga
        [57].S.BITS1.0   // 7-CON-1080 Enable
        [17].S.BITS1.0   // 7-ELV-1017 Enable
        [57].S.BITS1.1   // 7-CON-1080 Falla Resumen
        [57].S.BITS1.26   // 90-MMA-002 FLL
        [57].S.BITS1.27   // 90-MMA-002 FV0
        [57].S.BITS1.28   // 90-MMA-002 FATO
        [57].S.BITS2.20   // 7-CON-1080 Reset Falla
        [57].S.BITS2.23   // 7-CON-1080 Test
        [57].S.BITS2.27   // 7-CON-1080 Cmd. Open
        [57].S.BITS2.30   // 7-CON-1080 OUT CLOSE
        [58].S.BITS1.0   // 60-MRO-001-a Enable
        [58].S.BITS1.9   // TV-2 LM
        [58].S.BITS1.10   // TV-2 LH
        [58].S.BITS1.26   // 60-MRO-001-a FLL
        [58].S.BITS1.27   // 60-MRO-001-a FV0
        [179].S.BITS1.10   // TOL-064-00 LH
        [17].S.BITS1.29   // 90-CAN-004 Falla Abrir
        [17].S.BITS2.20   // 7-ELV-1017 Reset Falla
        [17].S.BITS2.23   // 7-ELV-1017 Test
        [136].S.BITS1.8   // BIN-34 LL
        [13].S.BITS1.8   // 90-TDC-001 Atollo
        [31].S.BITS1.4   // 7-RED-1052 Cmd. Automatico
        [41].S.BITS1.4   // 7-MMA-1065 Cmd. Automatico
        [77]   // 70-BIF-001
        [77].S.BITS1.0   // 7-RED-1090 Enable
        [77].S.BITS1.1   // 7-RED-1090 Falla Resumen
        [77].S.BITS1.4   // 7-RED-1090 Cmd. Automatico
        [77].S.BITS1.8   // ELE-608-00 IAto
        [21].S.BITS1.9   // 90-CAN-008 Conf. Cerrado
        [77].S.BITS1.10   // ELE-608-00 IV0
        [77].S.BITS2.11   // ELE-608-00 Enc Ext
        [77].S.BITS2.20   // 7-RED-1090 Reset Falla
        [77].S.BITS2.23   // 7-RED-1090 Test
        [77].S.BITS2.27   // 7-RED-1090 Cmd. Marcha
        [77].S.BITS2.30   // 7-RED-1090 OUT MARCHA
        [77].S.BITS2.31   // 70-BIF-001 Out Derecha
        [78].S.BITS1.0   // 7-RED-1091 Enable
        [78].S.BITS1.1   // 7-RED-1091 Falla Resumen
        [78].S.BITS1.2   // 7-RED-1091 Conf. Marcha
        [78].S.BITS1.4   // 7-RED-1091 Cmd. Automatico
        [78].S.BITS1.8   // BIN-05 LL
        [78].S.BITS1.9   // BIN-05 LM
        [78].S.BITS1.10   // BIN-05 LH
        [78].S.BITS1.26   // 7-RED-1091 FLL
        [78].S.BITS1.27   // 7-RED-1091 FV0
        [78].S.BITS1.28   // 7-RED-1091 FATO
        [78].S.BITS1.30   // 7-RED-1091 Falla Partida
        [78].S.BITS2.20   // 7-RED-1091 Reset Falla
        [78].S.BITS2.23   // 7-RED-1091 Test
        [78].S.BITS2.27   // 7-RED-1091 Cmd. Marcha
        [78].S.BITS2.30   // 7-RED-1091 OUT MARCHA
        [79].S.BITS1.0   // 7-ELV-1092 Enable
        [79].S.BITS1.1   // 7-ELV-1092 Falla Resumen
        [79].S.BITS1.2   // 7-ELV-1092 Conf. Marcha
        [79].S.BITS1.4   // 7-ELV-1092 Cmd. Automatico
        [79].S.BITS1.8   // RED-610-00 IAto
        [79].S.BITS1.10   // RED-610-00 IV0
        [15].S.BITS1.10   // 90-CAN-002 Conf. Abierto
        [79].S.BITS1.29   // 70-CAN-004 Falla Abrir
        [79].S.BITS2.11   // RED-610-00 Enc Ext
        [79].S.BITS2.20   // 7-ELV-1092 Reset Falla
        [79].S.BITS2.23   // 7-ELV-1092 Test
        [60].S.BITS1.0   // CV-4 Enable
        [4].S.BITS1.4   // 7-RED-1004 Cmd. Automatico
        [58].S.BITS1.28   // 60-MRO-001-a FATO
        [136].S.BITS2.31   // 100-CAN-003 OUT OPEN
        [5].S.BITS1.4   // 7-RED-1005 Cmd. Automatico
        [18].S.BITS1.0   // 7-BIF-1018 Enable
        [18].S.BITS2.20   // 7-BIF-1018 Reset Falla
        [18].S.BITS2.23   // 7-BIF-1018 Test
        [46].S.BITS1.9   // 90-MMA-001 Sobrecarga
        [49].S.BITS1.9   // 90-TOR-001 Sobrecarga
        [106].S.BITS1.2   // 7-ROS-1105 Conf. Marcha
        [1].S.BITS1.0   // 7-LMG-1001 Enable
        [22].S.BITS1.9   // 90-CAN-009 Conf. Cerrado
        [1].S.BITS1.1   // 7-LMG-1001 Falla Resumen
        [13].S.BITS1.10   // 90-TDC-001 Velocidad Cero
        [1].S.BITS1.2   // 7-LMG-1001 Conf. Marcha
        [102].S.BITS1.8   // 90-FIL-004 Atollo
        [127].S.BITS2.27   // 100-CAN-020 Cmd. Open
        [171].S.BITS1.27   // 7-VRT-1169 FV0
        [58].S.BITS2.23   // 60-MRO-001-a Test
        [50].S.BITS1.9   // 90-TAB-002 Sobrecarga
        [244].S.BITS1.8   // 100-TOR-020 Atollo
        [73].S.BITS1.9   // 90-MRO-002-A Sobrecarga
        [79].S.BITS2.31   // 70-CAN-004 OUT OPEN
        [19].S.BITS1.10   // 90-CAN-006 Conf. Abierto
        [303].S.BITS1.8   // XY-6170 Atollo
        [93].S.BITS1.26   // TCS-44_M FLL
        [137].S.BITS1.8   // RED-694-00 IAto
        [570].S.BITS2.31   // CV-12 OUT OPEN
        [103].S.BITS1.8   // 7-BIN-1102 LL
        [137].S.BITS1.26   // RIB-34 FLL
        [106].S.BITS1.29   // 70-CAN-21 Falla Abrir
        [23].S.BITS1.9   // 90-CAN-010 Conf. Cerrado
        [20].S.BITS1.7   // TOLV-001 LLL
        [74].S.BITS1.9   // 90-MRO-002-B Sobrecarga
        [197].S.BITS2.7   // MAG-034-01 Disable Codes
        [681].S.BITS1.10   // 120-BIN-031 LH
        [20].S.BITS1.8   // TOLV-001 LL
        [6].S.BITS1.4   // 7-COM-1006 Conf Pos Cerrar
        [54].S.BITS1.9   // 90-ALI-002 Sobrecarga
        [137].S.BITS1.27   // RIB-34 FV0
        [20].S.BITS1.9   // 90-CAN-007 Conf. Cerrado
        [137].S.BITS1.28   // RIB-34 FATO
        [24].S.BITS1.9   // 90-CAN-011 Conf. Cerrado
        [102].S.BITS1.9   // 90-FIL-004 Sobrecarga
        [48].S.BITS2.31   // CV-3 OUT OPEN
        [137].S.BITS2.11   // RED-694-00 Enc Ext
        [246].S.BITS1.8   // 100-TOR-019 Atollo
        [56].S.BITS1.9   // 90-VEN-002 Sobrecarga
        [44].S.BITS1.9   // 7-TV-107X LM
        [127].S.BITS2.30   // 100-CAN-020 OUT CLOSE
        [560].S.BITS2.23   // CV-11 Test
        [560].S.BITS1.0   // CV-11 Enable
        [7].S.BITS1.4   // 7-COM-1007 Conf Pos Cerrar
        [248].S.BITS1.8   // 100-TOR-018 Atollo
        [250].S.BITS1.8   // 100-TOR-017 Atollo
        [63].S.BITS1.8   // 90-MRO-001-A Atollo
        [58].S.BITS2.30   // 60-MRO-001-a OUT MARCHA
        [64].S.BITS1.8   // 90-MRO-001-B Atollo
        [93].S.BITS1.27   // TCS-44_M FV0
        [305].S.BITS1.8   // 8-TOL-608 LL
        [75].S.BITS1.9   // 90-MRO-002-C Sobrecarga
        [306].S.BITS1.8   // XY-6121 Atollo
        [104].S.BITS1.8   // 90-TDC-003 Atollo
        [309].S.BITS1.8   // XY-6100 Atollo
        [80].S.BITS1.0   // 7-RED-1093 Enable
        [683].S.BITS1.10   // 120-BIN-032 LH
        [203].S.BITS1.1   // 70-TOR-026 Falla Resumen
        [570].S.BITS2.23   // CV-12 Test
        [21].S.BITS1.7   // TOLV-002 LLL
        [21].S.BITS1.8   // TOLV-002 LL
        [171].S.BITS1.28   // 7-VRT-1169 FATO
        [102].S.BITS1.10   // 90-FIL-004 Velocidad Cero
        [138]   // 60-TOL-015-M
        [65].S.BITS1.8   // 7-BIN-1084 LL
        [313].S.BITS1.8   // XY-6102 Atollo
        [105].S.BITS1.8   // 7-BIN-1104 LL
        [22].S.BITS1.7   // TOLV-003 LLL
        [22].S.BITS1.8   // TOLV-003 LL
        [8].S.BITS1.4   // 7-COM-1008 Conf Pos Cerrar
        [138].S.BITS1.2   // CON-695-00 Open
        [23].S.BITS1.7   // TOLV-004 LLL
        [138].S.BITS1.4   // CON-695-00 Close
        [23].S.BITS2.11   // RED-648-00 Enc Ext
        [18].S.BITS1.8   // 90-TDC-002 Atollo
        [55].S.BITS1.9   // 90-FIL-002 Conf. Cerrado
        [677].S.BITS1.8   // 120-BIN-029 LL
        [677].S.BITS1.9   // 120-BIN-029 LM
        [679].S.BITS1.8   // 120-BIN-030 LL
        [106].S.BITS1.8   // 90-ELV-001 Atollo
        [24].S.BITS1.7   // TOLV-005 LLL
        [80].S.BITS1.1   // 7-RED-1093 Falla Resumen
        [80].S.BITS1.4   // 7-RED-1093 Cmd. Automatico
        [80].S.BITS1.8   // BIN-06 LL
        [80].S.BITS1.9   // BIN-06 LM
        [73].S.BITS1.8   // 90-MRO-002-A Atollo
        [16].S.BITS1.10   // 90-CAN-003 Conf. Abierto
        [24].S.BITS1.8   // TOLV-005 LL
        [138].S.BITS1.8   // BIN-35 LL
        [138].S.BITS1.9   // BIN-35 LM
        [26].S.BITS1.8   // 90-VEN-005 Atollo
        [93].S.BITS1.28   // TCS-44_M FATO
        [80].S.BITS1.10   // BIN-06 LH
        [24].S.BITS1.10   // 90-CAN-011 Conf. Abierto
        [679].S.BITS1.9   // 120-BIN-030 LM
        [25].S.BITS1.9   // CON-650-00 IClose
        [25].S.BITS1.10   // CON-650-00 IOpen
        [570].S.BITS1.0   // CV-12 Enable
        [18].S.BITS1.10   // 90-TDC-002 Velocidad Cero
        [138].S.BITS1.10   // BIN-35 LH
        [138].S.BITS2.7   // CON-695-00 Disable Codes
        [26].S.BITS1.0   // 7-CON-1026 Enable
        [138].S.BITS2.27   // 60-TOL-015-M Cmd
        [26].S.BITS1.26   // 90-VEN-005 FLL
        [26].S.BITS1.27   // 90-VEN-005 FV0
        [77].S.BITS1.30   // 7-RED-1090 Falla Partida
        [28].S.BITS1.8   // 7-TOL-1049 LL
        [9].S.BITS1.4   // 7-COM-1009 Conf Pos Cerrar
        [138].S.BITS2.31   // CON-695-00_Out
        [173].S.BITS1.0   // 70-TOR-017 Enable
        [10].S.BITS2.7   // BIF-698-00 Disable Codes
        [139].S.BITS1.0   // RIB-35 Enable
        [158].S.BITS1.7   // 70-BIN-010 LLL
        [158].S.BITS1.8   // 7-BIN-1157 LL
        [26].S.BITS1.28   // 90-VEN-005 FATO
        [26].S.BITS2.20   // 7-CON-1026 Reset Falla
        [26].S.BITS2.23   // 7-CON-1026 Test
        [103].S.BITS1.9   // 7-BIN-1102 LM
        [60].S.BITS1.8   // RED-658-00 IAto
        [60].S.BITS1.10   // RED-658-00 IV0
        [60].S.BITS2.11   // RED-658-00 Enc Ext
        [60].S.BITS2.27   // CV-4 Cmd. Open
        [158].S.BITS2.11   // ROS-014-00 Enc Ext
        [107].S.BITS1.8   // 7-BIN-1106 LL
        [17].S.BITS1.10   // 90-CAN-004 Conf. Abierto
        [97].S.BITS1.9   // 7-TOL-799 LM
        [103].S.BITS1.10   // 7-BIN-1102 LH
        [159].S.BITS1.8   // TOL-003-00 LL
        [159].S.BITS1.26   // 7-ROS-1158 FLL
        [159].S.BITS1.27   // 7-ROS-1158 FV0
        [159].S.BITS1.28   // 7-ROS-1158 FATO
        [159].S.BITS1.30   // 7-ROS-1158 Falla Partida
        [299].S.BITS1.9   // 100-TDP-006 Sobrecarga
        [29].S.BITS1.8   // 90-TDC-005 Atollo
        [60].S.BITS2.31   // CV-4 OUT OPEN
        [252].S.BITS1.8   // 100-TOR-016 Atollo
        [26].S.BITS2.27   // 7-CON-1026 Cmd. Open
        [303].S.BITS1.10   // XY-6170 Velocidad Cero
        [305].S.BITS1.10   // 8-TOL-608 LH
        [14].S.BITS1.2   // 7-CON-1014 Conf Pos Abrir
        [180].S.BITS1.2   // ROS-066-00 Run
        [306].S.BITS1.10   // XY-6121 Velocidad Cero
        [139].S.BITS1.1   // RIB-35 Falla Resumen
        [26].S.BITS2.30   // 7-CON-1026 OUT CLOSE
        [289].S.BITS1.8   // 100-TDP-003 Atollo
        [93].S.BITS1.30   // TCS-44_M Falla Partida
        [74].S.BITS1.8   // 90-MRO-002-B Atollo
        [151].S.BITS1.0   // 7-CON-1151 Enable
        [173].S.BITS1.1   // 70-TOR-017 Falla Resumen
        [84].S.BITS1.2   // 7-CON-1097 Conf Pos Abrir
        [93].S.BITS2.11   // RED-617-00 Enc Ext
        [139].S.BITS1.2   // RIB-35 Conf. Marcha
        [108].S.BITS1.0   // 7-ROS-1107 Enable
        [139].S.BITS1.4   // RIB-35 Cmd. Automatico
        [180].S.BITS1.7   // CV-006 LLL
        [26].S.BITS1.10   // 90-VEN-005 Velocidad Cero
        [108].S.BITS1.1   // 7-ROS-1107 Falla Resumen
        [27].S.BITS1.0   // 7-BIF-1027 Enable
        [93].S.BITS2.20   // TCS-44_M Reset Falla
        [15].S.BITS2.7   // CON-641-00 Disable Codes
        [173].S.BITS1.2   // 70-TOR-017 Conf. Marcha
        [16].S.BITS1.2   // 7-LMG-1016 Conf. Marcha
        [16].S.BITS2.7   // CON-642-00 Disable Codes
        [27].S.BITS1.26   // 60-FIL-003FLL
        [31].S.BITS1.30   // 7-RED-1052 Falla Partida
        [108].S.BITS1.2   // 7-ROS-1107 Conf. Marcha
        [108].S.BITS1.4   // 7-ROS-1107 Cmd. Automatico
        [173].S.BITS1.4   // 70-TOR-017 Cmd. Automatico
        [139].S.BITS1.9   // CON-696-00 IClose
        [27].S.BITS1.27   // 60-FIL-003FV0
        [17].S.BITS1.2   // 7-ELV-1017 Conf. Marcha
        [108].S.BITS1.26   // 7-ROS-1107 FLL
        [139].S.BITS1.10   // CON-696-00 IOpen
        [108].S.BITS1.27   // 7-ROS-1107 FV0
        [180].S.BITS2.11   // ROS-066-00 Enc Ext
        [165].S.BITS1.8   // TOL-006-00 LL
        [108].S.BITS1.28   // 7-ROS-1107 FATO
        [108].S.BITS1.30   // 7-ROS-1107 Falla Partida
        [80].S.BITS1.29   // 70-CAN-005 Falla Abrir
        [180].S.BITS2.27   // ROS-066-00 Cmd
        [180].S.BITS2.31   // ROS-066-00 Out
        [108].S.BITS2.11   // RED-623-00 Enc Ext
        [27].S.BITS1.28   // 60-FIL-003FATO
        [17].S.BITS2.7   // CON-643-00 Disable Codes
        [108].S.BITS1.8   // 90-ELV-003 Atollo
        [27].S.BITS2.20   // 7-BIF-1027 Reset Falla
        [27].S.BITS2.23   // 7-BIF-1027 Test
        [84].S.BITS1.29   // 7-CON-1097 Falla Abrir
        [159].S.BITS2.30   // 7-ROS-1158 OUT MARCHA
        [40].S.BITS1.8   // 90-TAB-001 Atollo
        [309].S.BITS1.10   // XY-6100 Velocidad Cero
        [313].S.BITS1.10   // XY-6102 Velocidad Cero
        [93].S.BITS2.23   // TCS-44_M Test
        [128].S.BITS1.8   // BIN-30 LL
        [84].S.BITS2.11   // ESP-613-00 Enc Ext
        [20].S.BITS1.10   // 90-CAN-007 Conf. Abierto
        [139].S.BITS1.26   // RIB-35 FLL
        [93].S.BITS2.27   // TCS-44_M Cmd. Marcha
        [160].S.BITS1.2   // ROS-015-00 Run
        [93].S.BITS2.30   // TCS-44_M OUT MARCHA
        [28].S.BITS1.10   // 7-TOL-1049 LH
        [53].S.BITS1.4   // 7-RED-1076 Cmd. Automatico
        [132].S.BITS1.8   // BIN-32 LL
        [21].S.BITS1.10   // 90-CAN-008 Conf. Abierto
        [18].S.BITS2.7   // CON-644-00 Disable Codes
        [235].S.BITS1.8   // Nivel Vacio Estanque Faenadora
        [139].S.BITS1.27   // RIB-35 FV0
        [165].S.BITS1.26   // 7-ROS-1164 FLL
        [19].S.BITS2.7   // CON-645-00 Disable Codes
        [108].S.BITS2.20   // 7-ROS-1107 Reset Falla
        [681].S.BITS1.8   // 120-BIN-031 LL
        [109].S.BITS1.8   // 7-BIN-1108 LL
        [28].S.BITS1.7   // 60-TOL-003 LLL
        [165].S.BITS1.27   // 7-ROS-1164 FV0
        [20].S.BITS2.7   // CON-646-00 Disable Codes
        [104].S.BITS1.10   // 90-TDC-003 Velocidad Cero
        [21].S.BITS2.7   // CON-647-00 Disable Codes
        [54].S.BITS1.4   // 7-CON-1077 Conf Pos Cerrar
        [108].S.BITS2.23   // 7-ROS-1107 Test
        [75].S.BITS1.8   // 90-MRO-002-C Atollo
        [139].S.BITS1.28   // RIB-35 FATO
        [108].S.BITS2.27   // 7-ROS-1107 Cmd. Marcha
        [24].S.BITS2.7   // CON-649-00 Disable Codes
        [55].S.BITS1.4   // 7-RED-1078 Cmd. Automatico
        [108].S.BITS2.30   // 7-ROS-1107 OUT MARCHA
        [181].S.BITS1.7   // CV-007 LLL
        [83].S.BITS1.9   // 90-MRO-003-A Sobrecarga
        [678].S.BITS2.23   // 120-CAN-067 Test
        [29].S.BITS1.7   // 60-TOL-002 LLL
        [31].S.BITS1.1   // 7-RED-1052 Falla Resumen
        [37].S.BITS1.4   // 60-VEN-004A Cmd. Automatico
        [83].S.BITS1.8   // 90-MRO-003-A Atollo
        [25].S.BITS2.7   // CON-650-00 Disable Codes
        [101].S.BITS1.29   // 70-BIF-003 Falla Pos. Izquierda
        [26].S.BITS1.30   // 7-CON-1026 Falla Cerrar
        [30].S.BITS1.7   // 60-TOL-001 LLL
        [30].S.BITS1.8   // 60-TOL-001 LL
        [30].S.BITS1.9   // 60-TOL-001 LM
        [30].S.BITS1.10   // 60-TOL-001 LH
        [30].S.BITS2.31   // CON-655-00_Out
        [31].S.BITS1.0   // 7-RED-1052 Enable
        [31].S.BITS1.26   // 7-RED-1052 FLL
        [31].S.BITS1.27   // 7-RED-1052 FV0
        [31].S.BITS1.28   // 7-RED-1052 FATO
        [31].S.BITS2.23   // 7-RED-1052 Test
        [32].S.BITS1.0   // 7-RED-1053 Enable
        [32].S.BITS1.8   // 90-TOL-002 LL
        [32].S.BITS1.9   // 90-TOL-002 LM
        [32].S.BITS1.10   // 90-TOL-002 LH
        [32].S.BITS1.29   // 60-CAN-015 Falla Abrir
        [32].S.BITS2.20   // 7-RED-1053 Reset Falla
        [32].S.BITS2.23   // 7-RED-1053 Test
        [33].S.BITS1.0   // 7-CON-1054 Enable
        [33].S.BITS1.26   // 60-ALI-004 FLL
        [139].S.BITS1.30   // RIB-35 Falla Partida
        [33].S.BITS1.27   // 60-ALI-004 FV0
        [171].S.BITS1.30   // 7-VRT-1169 Falla Partida
        [139].S.BITS2.7   // CON-696-00 Disable Codes
        [94].S.BITS1.0   // TCS-44 Enable
        [101].S.BITS2.26   // 70-BIF-003 Cmd. Pos . Izquierda
        [84].S.BITS1.9   // 90-MRO-003-B Sobrecarga
        [94].S.BITS1.1   // TCS-44 Falla Resumen
        [316].S.BITS1.8   // 8-ENF-630 LL
        [41].S.BITS1.1   // 7-MMA-1065 Falla Resumen
        [203].S.BITS1.2   // 70-TOR-026 Conf. Marcha
        [47].S.BITS1.4   // 7-ELV-1070 Cmd. Automatico
        [173].S.BITS1.8   // TOL-010-00 LL
        [85].S.BITS1.9   // 90-MRO-003-C Sobrecarga
        [128].S.BITS2.11   // ELE-635-00 Enc Ext
        [112].S.BITS1.9   // 100-FIL-001 Sobrecarga
        [57].S.BITS1.9   // 90-MMA-002 Sobrecarga
        [59].S.BITS1.9   // 7-BIN-1081 LM
        [153].S.BITS1.26   // 70-TOR-008 FLL
        [680].S.BITS2.23   // 120-CAN-068 Test
        [26].S.BITS2.7   // CON-651-00 Disable Codes
        [62].S.BITS1.9   // 90-ALI-003 Sobrecarga
        [43].S.BITS1.8   // 90-ALI-001 Atollo
        [317].S.BITS1.8   // 100-VEN-COLINA-1 Atollo
        [85].S.BITS1.2   // 90-MRO-003-C Conf. Marcha
        [72].S.BITS1.9   // 90-ALI-004 Sobrecarga
        [165].S.BITS1.28   // 7-ROS-1164 FATO
        [82].S.BITS1.9   // 90-ALI-005 Sobrecarga
        [292].S.BITS1.8   // 100-TDP-004 Atollo
        [118]   // 70-BIF-002
        [29].S.BITS1.10   // 90-TDC-005 Velocidad Cero
        [85].S.BITS1.10   // 90-MRO-003-C Velocidad Cero
        [85].S.BITS1.29   // 70-CAN-008 Falla Abrir
        [351].S.BITS1.9   // 110-TOR-005 Sobrecarga
        [139].S.BITS2.20   // RIB-35 Reset Falla
        [45].S.BITS1.8   // 90-VEN-001 Atollo
        [153].S.BITS1.27   // 70-TOR-008 FV0
        [147].S.BITS1.27   // 70-TOR-004 FV0
        [85].S.BITS2.11   // VEN-613-01 Enc Ext
        [27].S.BITS2.7   // CON-652-00 Disable Codes
        [28].S.BITS2.7   // CON-653-00 Disable Codes
        [29].S.BITS2.7   // CON-654-00 Disable Codes
        [113].S.BITS1.9   // 7-BIN-1112 LM
        [115].S.BITS1.9   // 7-BIN-1114 LM
        [92].S.BITS1.9   // 7-TOL-797 LM
        [93].S.BITS1.9   // 90-FIL-003 Sobrecarga
        [30].S.BITS2.7   // CON-655-00 Disable Codes
        [96].S.BITS1.9   // 7-TOL-798 LM
        [31].S.BITS2.30   // 7-RED-1052 OUT MARCHA
        [33].S.BITS1.28   // 60-ALI-004 FATO
        [118].S.BITS1.8   // BIN-25 LL
        [118].S.BITS1.9   // BIN-25 LM
        [139].S.BITS2.23   // RIB-35 Test
        [33].S.BITS1.30   // 7-CON-1054 Falla Cerrar
        [94].S.BITS1.2   // TCS-44 Conf. Marcha
        [94].S.BITS1.4   // TCS-44 Cmd. Automatico
        [35].S.BITS1.2   // 7-CON-1055 Conf Pos Abrir
        [86].S.BITS1.0   // tcs-28_M Enable
        [86].S.BITS1.1   // tcs-28_M Falla Resumen
        [86].S.BITS1.2   // tcs-28_M Conf. Marcha
        [86].S.BITS1.4   // tcs-28_M Cmd. Automatico
        [86].S.BITS1.8   // BIN-09 LL
        [352].S.BITS1.9   // 110-TDC-002 Sobrecarga
        [132].S.BITS2.11   // RED-690-00 Enc Ext
        [116].S.BITS1.9   // 100-ELV-001 Sobrecarga
        [86].S.BITS1.9   // BIN-09 LM
        [86].S.BITS1.10   // BIN-09 LH
        [151].S.BITS1.1   // 7-CON-1151 Falla Resumen
        [86].S.BITS1.29   // 70-CAN-009 Falla Abrir
        [86].S.BITS1.30   // tcs-28_M Falla Partida
        [118].S.BITS1.10   // BIN-25 LH
        [36].S.BITS1.30   // 60-VEN-002 Falla Partida
        [37].S.BITS1.1   // 60-VEN-004A Falla Resumen
        [94].S.BITS1.26   // TCS-44 FLL
        [94].S.BITS1.27   // TCS-44 FV0
        [33].S.BITS2.20   // 7-CON-1054 Reset Falla
        [139].S.BITS2.27   // RIB-35 Cmd. Marcha
        [118].S.BITS1.29   // CV-8 Falla Abrir
        [118].S.BITS2.7   // CON-628-00Cmd Open
        [86].S.BITS2.20   // tcs-28_M Reset Falla
        [293].S.BITS1.8   // 100-ELV-002 Atollo
        [22].S.BITS1.10   // 90-CAN-009 Conf. Abierto
        [33].S.BITS2.23   // 7-CON-1054 Test
        [129].S.BITS1.0   // RIB-30 Enable
        [118].S.BITS2.26   // 70-BIF-002 Cmd. Pos . Izquierda
        [86].S.BITS2.23   // tcs-28_M Test
        [94].S.BITS1.28   // TCS-44 FATO
        [173].S.BITS1.9   // TOL-010-00 LM
        [153].S.BITS1.28   // 70-TOR-008 FATO
        [118].S.BITS2.31   // CV-8 OUT OPEN
        [38].S.BITS1.4   // 60-TOR-002Cmd. Automatico
        [33].S.BITS2.27   // 7-CON-1054 Cmd. Open
        [119].S.BITS1.0   // 70-TDC-005 Enable
        [160].S.BITS1.7   // 70-BIN-011 LLL
        [86].S.BITS2.27   // tcs-28_M Cmd. Marcha
        [33].S.BITS2.30   // 7-CON-1054 OUT CLOSE
        [34].S.BITS1.0   // 7-BIF-1055 Enable
        [34].S.BITS1.9   // 90-TOL-004 LM
        [139].S.BITS2.30   // RIB-35 OUT MARCHA
        [34].S.BITS1.10   // 90-TOL-004 LH
        [40].S.BITS1.10   // 90-TAB-001 Velocidad Cero
        [39].S.BITS1.30   // 60-TOR-002 Falla Partida
        [129].S.BITS1.1   // RIB-30 Falla Resumen
        [382].S.BITS1.8   // 110-ENF-001/1-4 Atollo
        [153].S.BITS1.30   // 7-CON-1153 Falla Cerrar
        [34].S.BITS1.26   // 60-MMA-002 FLL
        [109].S.BITS1.2   // 90-ELV-004 Conf. Marcha
        [384].S.BITS1.8   // 110-ENF-001/1-1 Atollo
        [129].S.BITS1.2   // RIB-30 Conf. Marcha
        [389].S.BITS1.8   // 110-VAL-001/1-1 Atollo
        [40].S.BITS1.30   // 7-VRT-1064 Falla Partida
        [43].S.BITS1.10   // 90-ALI-001 Velocidad Cero
        [191].S.BITS1.9   // CON-030-00IClose
        [390].S.BITS1.8   // 110-VEN-001/1-1 Atollo
        [34].S.BITS1.27   // 60-MMA-002 FV0
        [129].S.BITS1.4   // RIB-30 Cmd. Automatico
        [160].S.BITS1.8   // 7-BIN-1159 LL
        [140].S.BITS1.7   // 70-BIN-001 LLL
        [94].S.BITS1.30   // TCS-44 Falla Partida
        [94].S.BITS2.7   // CON-699-00 Disable Codes
        [129].S.BITS1.8   // 7-BIN-1128 LL
        [94].S.BITS2.20   // TCS-44 Reset Falla
        [43].S.BITS1.30   // 7-VEN-1067 Falla Partida
        [140].S.BITS1.8   // 70-BIN-001 LL
        [129].S.BITS1.10   // 7-BIN-1128 LH
        [46].S.BITS1.8   // 90-MMA-001 Atollo
        [94].S.BITS2.23   // TCS-44 Test
        [129].S.BITS1.26   // RIB-30 FLL
        [153].S.BITS2.27   // 7-CON-1153 Cmd. Open
        [94].S.BITS2.27   // TCS-44 Cmd. Marcha
        [86].S.BITS2.30   // tcs-28_M OUT MARCHA
        [98].S.BITS1.9   // 7-ELV-100 LM
        [105].S.BITS1.10   // 7-BIN-1104 LH
        [322].S.BITS1.8   // 100-MIX-001-M Atollo
        [140].S.BITS1.9   // 70-BIN-001 LM
        [163].S.BITS1.8   // BINMICROA-2 LL
        [140].S.BITS1.10   // 70-BIN-001 LH
        [140].S.BITS2.7   // CON-697-00 Disable Codes
        [58].S.BITS1.4   // 60-MRO-001-a Cmd. Automatico
        [94].S.BITS2.30   // TCS-44 OUT MARCHA
        [109].S.BITS1.29   // 70-CAN-11 Falla Abrir
        [391].S.BITS1.8   // 110-ENF-001/1-5 Atollo
        [34].S.BITS1.28   // 60-MMA-002 FATO
        [153].S.BITS2.30   // 7-CON-1153 OUT CLOSE
        [54].S.BITS1.30   // 7-CON-1077 Falla Cerrar
        [94].S.BITS2.31   // CON-699-00_Out
        [34].S.BITS2.7   // CON-659-01Cmd Open
        [106].S.BITS1.10   // 90-ELV-001 Velocidad Cero
        [154].S.BITS1.7   // 70-BIN-008 LLL
        [95].S.BITS1.0   // CV-7 Enable
        [34].S.BITS2.20   // 7-BIF-1055 Reset Falla
        [34].S.BITS2.23   // 7-BIF-1055 Test
        [86].S.BITS2.31   // 70-CAN-009 OUT OPEN
        [140].S.BITS2.31   // CON-697-00_Out
        [294].S.BITS1.8   // 100-TDP-005 Atollo
        [122].S.BITS1.9   // 100-TDP-001 Sobrecarga
        [35].S.BITS1.0   // 7-CON-1055 Enable
        [35].S.BITS1.9   // 90-TOL-005 LM
        [35].S.BITS1.10   // 90-TOL-005 LH
        [119].S.BITS1.1   // 70-TDC-005 Falla Resumen
        [35].S.BITS1.26   // 60-FIL-002FLL
        [681].S.BITS1.9   // 120-BIN-031 LM
        [62].S.BITS1.29   // 60-FIL-004 Falla Abrir
        [402].S.BITS1.8   // 110-ENF-002/1-4 Atollo
        [365].S.BITS1.8   // 110-CAN-010/1 Atollo
        [35].S.BITS1.27   // 60-FIL-002FV0
        [35].S.BITS1.28   // 60-FIL-002FATO
        [154].S.BITS1.8   // 70-BIN-008 LL
        [370].S.BITS1.8   // 110-TOR-001/1 Atollo
        [44].S.BITS1.30   // 90-FIL-001 Falla Cerrar
        [80].S.BITS2.7   // CON-611-00 Disable Codes
        [404].S.BITS1.8   // 110-ENF-002/1-1 Atollo
        [141].S.BITS1.0   // 7-ROS-1140 Enable
        [682].S.BITS2.23   // 120-CAN-069 Test
        [141].S.BITS1.1   // 7-ROS-1140 Falla Resumen
        [95].S.BITS1.1   // CV-7 Falla Resumen
        [141].S.BITS1.2   // 7-ROS-1140 Conf. Marcha
        [35].S.BITS1.29   // 7-CON-1055 Falla Abrir
        [141].S.BITS1.4   // 7-ROS-1140 Cmd. Automatico
        [49].S.BITS1.8   // 90-TOR-001 Atollo
        [35].S.BITS2.7   // CON-659-00Cmd Open
        [173].S.BITS1.10   // TOL-010-00 LH
        [173].S.BITS1.26   // 70-TOR-017 FLL
        [141].S.BITS1.26   // 7-ROS-1140 FLL
        [156].S.BITS1.7   // 70-BIN-009 LLL
        [45].S.BITS1.2   // 7-ROS-1068 Conf. Marcha
        [45].S.BITS2.7   // CON-665-00 Disable Codes
        [191].S.BITS1.10   // CON-030-00IOpen
        [185].S.BITS1.8   // TOL-025-00 LL
        [58].S.BITS1.1   // 60-MRO-001-a Falla Resumen
        [147].S.BITS1.28   // 70-TOR-004 FATO
        [35].S.BITS2.20   // 7-CON-1055 Reset Falla
        [156].S.BITS1.8   // 7-BIN-1155 LL
        [151].S.BITS1.4   // 7-CON-1151 Conf Pos Cerrar
        [58].S.BITS1.30   // 60-MRO-001-a Falla Partida
        [35].S.BITS2.23   // 7-CON-1055 Test
        [35].S.BITS2.27   // 7-CON-1055 Cmd. Open
        [110].S.BITS1.2   // 7-ROS-1109 Conf. Marcha
        [160].S.BITS1.9   // 7-BIN-1159 LM
        [409].S.BITS1.8   // 110-VAL-002/1-1 Atollo
        [171].S.BITS2.20   // 7-VRT-1169 Reset Falla
        [129].S.BITS1.27   // RIB-30 FV0
        [410].S.BITS1.8   // 110-VEN-002/1-1 Atollo
        [35].S.BITS2.30   // 7-CON-1055 OUT CLOSE
        [160].S.BITS1.10   // 7-BIN-1159 LH
        [35].S.BITS2.31   // 7-CON-1055 OUT OPEN
        [36].S.BITS1.0   // 60-VEN-002 Enable
        [36].S.BITS1.9   // 7-BIN-1060 LM
        [411].S.BITS1.8   // 110-ENF-002/1-5 Atollo
        [110].S.BITS1.8   // BIN-21 LL
        [126].S.BITS1.9   // 100-TDP-002 Sobrecarga
        [160].S.BITS2.11   // ROS-015-00 Enc Ext
        [141].S.BITS1.27   // 7-ROS-1140 FV0
        [129].S.BITS1.28   // RIB-30 FATO
        [196].S.BITS2.11   // MAG-034-00 Enc Ext
        [171].S.BITS2.23   // 7-VRT-1169 Test
        [95].S.BITS1.2   // CV-7 Conf Pos Abrir
        [173].S.BITS1.27   // 70-TOR-017 FV0
        [141].S.BITS1.28   // 7-ROS-1140 FATO
        [110].S.BITS1.9   // BIN-21 LM
        [110].S.BITS1.10   // BIN-21 LH
        [141].S.BITS1.30   // 7-ROS-1140 Falla Partida
